LIN {X 0,Y 253.185,Z 308.196,A -85,B 0,C 180,E1 -19429.256,E2 -19429.256} C_VEL
LIN {X 0,Y 250.888,Z 304.72,A -85,B 0,C 180,E1 -19430.326,E2 -19430.326} C_VEL
LIN {X 0,Y 250.004,Z 303.462,A -85,B 0,C 180,E1 -19430.751,E2 -19430.751} C_VEL
LIN {X 0,Y 247.713,Z 300.458,A -85,B 0,C 180,E1 -19431.846,E2 -19431.846} C_VEL
LIN {X 0,Y 246.985,Z 298.947,A -85,B 0,C 180,E1 -19432.234,E2 -19432.234} C_VEL
LIN {X 0,Y 244.491,Z 296.754,A -85,B 0,C 180,E1 -19433.399,E2 -19433.399} C_VEL
LIN {X 0,Y 243.101,Z 294.193,A -85,B 0,C 180,E1 -19434.194,E2 -19434.194} C_VEL
LIN {X 0,Y 242.944,Z 293.571,A -85,B 0,C 180,E1 -19434.399,E2 -19434.399} C_VEL
LIN {X 0,Y 243.113,Z 292.905,A -85,B 0,C 180,E1 -19438.345,E2 -19438.345} C_VEL
LIN {X 0,Y 243.203,Z 292.718,A -85,B 0,C 180,E1 -19440.002,E2 -19440.002} C_VEL
LIN {X 0,Y 242.902,Z 292.579,A -85,B 0,C 180,E1 -19443.319,E2 -19443.319} C_VEL
LIN {X 0,Y 242.885,Z 292.698,A -85,B 0,C 180,E1 -19448.32,E2 -19448.32} C_VEL
LIN {X 0,Y 242.8,Z 293.112,A -85,B 0,C 180,E1 -19451.692,E2 -19451.692} C_VEL
LIN {X 0,Y 242.869,Z 293.758,A -85,B 0,C 180,E1 -19455.098,E2 -19455.098} C_VEL
LIN {X 0,Y 242.939,Z 294.698,A -85,B 0,C 180,E1 -19458.557,E2 -19458.557} C_VEL
LIN {X 0,Y 243.14,Z 296.031,A -85,B 0,C 180,E1 -19462.34,E2 -19462.34} C_VEL
LIN {X 0,Y 243.449,Z 297.883,A -85,B 0,C 180,E1 -19466.505,E2 -19466.505} C_VEL
LIN {X 0,Y 243.751,Z 299.841,A -85,B 0,C 180,E1 -19470.122,E2 -19470.122} C_VEL
LIN {X 0,Y 244.055,Z 301.816,A -85,B 0,C 180,E1 -19473.27,E2 -19473.27} C_VEL
LIN {X 0,Y 243.519,Z 302.82,A -85,B 0,C 180,E1 -19474.187,E2 -19474.187} C_VEL
LIN {X 0,Y 241.244,Z 305.585,A -85,B 0,C 180,E1 -19475.584,E2 -19475.584} C_VEL
LIN {X 0,Y 239.817,Z 308.232,A -85,B 0,C 180,E1 -19476.663,E2 -19476.663} C_VEL
LIN {X 0,Y 239.881,Z 310.193,A -85,B 0,C 180,E1 -19477.486,E2 -19477.486} C_VEL
LIN {X 0,Y 240.255,Z 310.779,A -85,B 0,C 180,E1 -19477.754,E2 -19477.754} C_VEL
LIN {X 0,Y 241.849,Z 312.454,A -85,B 0,C 180,E1 -19478.568,E2 -19478.568} C_VEL
LIN {X 0,Y 243.742,Z 316.37,A -85,B 0,C 180,E1 -19479.64,E2 -19479.64} C_VEL
LIN {X 0,Y 245.733,Z 319.174,A -85,B 0,C 180,E1 -19480.66,E2 -19480.66} C_VEL
LIN {X 0,Y 247.963,Z 323.482,A -85,B 0,C 180,E1 -19481.833,E2 -19481.833} C_VEL
LIN {X 0,Y 249.149,Z 325.386,A -85,B 0,C 180,E1 -19482.405,E2 -19482.405} C_VEL
LIN {X 0,Y 251.625,Z 330.796,A -85,B 0,C 180,E1 -19483.741,E2 -19483.741} C_VEL
LIN {X 0,Y 253.857,Z 336.868,A -85,B 0,C 180,E1 -19485.042,E2 -19485.042} C_VEL
LIN {X 0,Y 256.669,Z 347.947,A -85,B 0,C 180,E1 -19487.095,E2 -19487.095} C_VEL
LIN {X 0,Y 258.818,Z 360.728,A -85,B 0,C 180,E1 -19489.332,E2 -19489.332} C_VEL
LIN {X 0,Y 259.644,Z 370.662,A -85,B 0,C 180,E1 -19491.018,E2 -19491.018} C_VEL
LIN {X 0,Y 259.672,Z 381.634,A -85,B 0,C 180,E1 -19492.891,E2 -19492.891} C_VEL
LIN {X 0,Y 258.885,Z 392.631,A -85,B 0,C 180,E1 -19494.838,E2 -19494.838} C_VEL
LIN {X 0,Y 254.509,Z 405.491,A -85,B 0,C 180,E1 -19496.951,E2 -19496.951} C_VEL
LIN {X 0,Y 250.343,Z 416.596,A -85,B 0,C 180,E1 -19499.182,E2 -19499.182} C_VEL
LIN {X 0,Y 246.132,Z 427.508,A -85,B 0,C 180,E1 -19501.893,E2 -19501.893} C_VEL
LIN {X 0,Y 242.659,Z 436.647,A -85,B 0,C 180,E1 -19504.712,E2 -19504.712} C_VEL
LIN {X 0,Y 239.529,Z 444.307,A -85,B 0,C 180,E1 -19507.579,E2 -19507.579} C_VEL
LIN {X 0,Y 236.803,Z 451.549,A -85,B 0,C 180,E1 -19510.947,E2 -19510.947} C_VEL
LIN {X 0,Y 234.837,Z 457.354,A -85,B 0,C 180,E1 -19514.376,E2 -19514.376} C_VEL
LIN {X 0,Y 233.597,Z 461.841,A -85,B 0,C 180,E1 -19517.844,E2 -19517.844} C_VEL
LIN {X 0,Y 233.019,Z 465.103,A -85,B 0,C 180,E1 -19521.328,E2 -19521.328} C_VEL
LIN {X 0,Y 232.953,Z 467.185,A -85,B 0,C 180,E1 -19524.808,E2 -19524.808} C_VEL
LIN {X 0,Y 232.961,Z 468.034,A -85,B 0,C 180,E1 -19528.272,E2 -19528.272} C_VEL
LIN {X 0,Y 232.997,Z 468.019,A -85,B 0,C 180,E1 -19530.001,E2 -19530.001} C_VEL
LIN {X 0,Y 232.972,Z 467.09,A -85,B 0,C 180,E1 -19533.46,E2 -19533.46} C_VEL
LIN {X 0,Y 233.034,Z 465.926,A -85,B 0,C 180,E1 -19535.582,E2 -19535.582} C_VEL
LIN {X 0,Y 233.072,Z 463.412,A -85,B 0,C 180,E1 -19538.673,E2 -19538.673} C_VEL
LIN {X 0,Y 233.62,Z 459.368,A -85,B 0,C 180,E1 -19542.158,E2 -19542.158} C_VEL
LIN {X 0,Y 234.812,Z 453.934,A -85,B 0,C 180,E1 -19545.628,E2 -19545.628} C_VEL
LIN {X 0,Y 236.689,Z 446.986,A -85,B 0,C 180,E1 -19549.065,E2 -19549.065} C_VEL
LIN {X 0,Y 238.891,Z 439.482,A -85,B 0,C 180,E1 -19552.031,E2 -19552.031} C_VEL
LIN {X 0,Y 241.773,Z 430.492,A -85,B 0,C 180,E1 -19554.93,E2 -19554.93} C_VEL
LIN {X 0,Y 244.548,Z 421.312,A -85,B 0,C 180,E1 -19557.377,E2 -19557.377} C_VEL
LIN {X 0,Y 247.908,Z 410.531,A -85,B 0,C 180,E1 -19559.744,E2 -19559.744} C_VEL
LIN {X 0,Y 251.243,Z 398.782,A -85,B 0,C 180,E1 -19561.871,E2 -19561.871} C_VEL
LIN {X 0,Y 253.709,Z 390.137,A -85,B 0,C 180,E1 -19563.169,E2 -19563.169} C_VEL
LIN {X 0,Y 253.899,Z 385.833,A -85,B 0,C 180,E1 -19563.857,E2 -19563.857} C_VEL
LIN {X 0,Y 253.203,Z 373.399,A -85,B 0,C 180,E1 -19565.801,E2 -19565.801} C_VEL
LIN {X 0,Y 251.448,Z 358.938,A -85,B 0,C 180,E1 -19567.852,E2 -19567.852} C_VEL
LIN {X 0,Y 249.014,Z 346.189,A -85,B 0,C 180,E1 -19569.525,E2 -19569.525} C_VEL
LIN {X 0,Y 245.629,Z 332.569,A -85,B 0,C 180,E1 -19571.179,E2 -19571.179} C_VEL
LIN {X 0,Y 241.385,Z 319.106,A -85,B 0,C 180,E1 -19572.752,E2 -19572.752} C_VEL
LIN {X 0,Y 239.34,Z 314.218,A -85,B 0,C 180,E1 -19573.368,E2 -19573.368} C_VEL
LIN {X 0,Y 238.309,Z 310.845,A -85,B 0,C 180,E1 -19573.734,E2 -19573.734} C_VEL
LIN {X 0,Y 237.815,Z 307.272,A -85,B 0,C 180,E1 -19577.178,E2 -19577.178} C_VEL
LIN {X 0,Y 236.974,Z 303.106,A -85,B 0,C 180,E1 -19581.477,E2 -19581.477} C_VEL
LIN {X 0,Y 236.258,Z 298.657,A -85,B 0,C 180,E1 -19586.402,E2 -19586.402} C_VEL
LIN {X 0,Y 235.576,Z 294.467,A -85,B 0,C 180,E1 -19591.487,E2 -19591.487} C_VEL
LIN {X 0,Y 235.184,Z 291.61,A -85,B 0,C 180,E1 -19595.267,E2 -19595.267} C_VEL
LIN {X 0,Y 234.976,Z 290.842,A -85,B 0,C 180,E1 -19596.651,E2 -19596.651} C_VEL
LIN {X 0,Y 235.016,Z 290.835,A -85,B 0,C 180,E1 -19600.793,E2 -19600.793} C_VEL
LIN {X 0,Y 235.121,Z 290.825,A -85,B 0,C 180,E1 -19604.392,E2 -19604.392} C_VEL
LIN {X 0,Y 235.221,Z 290.812,A -85,B 0,C 180,E1 -19609.671,E2 -19609.671} C_VEL
LIN {X 0,Y 235.365,Z 290.793,A -85,B 0,C 180,E1 -19613.138,E2 -19613.138} C_VEL
LIN {X 0,Y 235.6,Z 290.764,A -85,B 0,C 180,E1 -19618.289,E2 -19618.289} C_VEL
LIN {X 0,Y 235.6,Z 290.761,A -85,B 0,C 180,E1 -19621.708,E2 -19621.708} C_VEL
LIN {X 0,Y 235.41,Z 290.784,A -85,B 0,C 180,E1 -19626.857,E2 -19626.857} C_VEL
LIN {X 0,Y 235.257,Z 290.798,A -85,B 0,C 180,E1 -19630.324,E2 -19630.324} C_VEL
LIN {X 0,Y 235.116,Z 290.82,A -85,B 0,C 180,E1 -19635.604,E2 -19635.604} C_VEL
LIN {X 0,Y 235.011,Z 290.825,A -85,B 0,C 180,E1 -19639.203,E2 -19639.203} C_VEL
LIN {X 0,Y 234.962,Z 290.84,A -85,B 0,C 180,E1 -19642.88,E2 -19642.88} C_VEL
LIN {X 0,Y 234.968,Z 290.832,A -85,B 0,C 180,E1 -19646.655,E2 -19646.655} C_VEL
LIN {X 0,Y 234.922,Z 290.845,A -85,B 0,C 180,E1 -19650.566,E2 -19650.566} C_VEL
LIN {X 0,Y 234.959,Z 290.832,A -85,B 0,C 180,E1 -19654.63,E2 -19654.63} C_VEL
LIN {X 0,Y 234.94,Z 290.843,A -85,B 0,C 180,E1 -19658.942,E2 -19658.942} C_VEL
LIN {X 0,Y 234.901,Z 290.836,A -85,B 0,C 180,E1 -19663.48,E2 -19663.48} C_VEL
LIN {X 0,Y 234.962,Z 290.841,A -85,B 0,C 180,E1 -19666.53,E2 -19666.53} C_VEL
LIN {X 0,Y 234.951,Z 290.84,A -85,B 0,C 180,E1 -19671.084,E2 -19671.084} C_VEL
LIN {X 0,Y 234.955,Z 290.834,A -85,B 0,C 180,E1 -19675.365,E2 -19675.365} C_VEL
LIN {X 0,Y 234.964,Z 290.836,A -85,B 0,C 180,E1 -19680.155,E2 -19680.155} C_VEL
LIN {X 0,Y 234.988,Z 290.838,A -85,B 0,C 180,E1 -19683.791,E2 -19683.791} C_VEL
LIN {X 0,Y 235.004,Z 290.833,A -85,B 0,C 180,E1 -19688.968,E2 -19688.968} C_VEL
LIN {X 0,Y 235.089,Z 290.822,A -85,B 0,C 180,E1 -19693.058,E2 -19693.058} C_VEL
LIN {X 0,Y 235.139,Z 290.818,A -85,B 0,C 180,E1 -19697.922,E2 -19697.922} C_VEL
LIN {X 0,Y 235.194,Z 290.863,A -85,B 0,C 180,E1 -19699.252,E2 -19699.252} C_VEL
LIN {X 0,Y 236.19,Z 293.619,A -85,B 0,C 180,E1 -19699.592,E2 -19699.592} C_VEL
LIN {X 0,Y 237.987,Z 295.971,A -85,B 0,C 180,E1 -19700.061,E2 -19700.061} C_VEL
LIN {X 0,Y 243.806,Z 306.338,A -85,B 0,C 180,E1 -19701.824,E2 -19701.824} C_VEL
LIN {X 0,Y 250.316,Z 320.248,A -85,B 0,C 180,E1 -19704.118,E2 -19704.118} C_VEL
LIN {X 0,Y 253.968,Z 333.092,A -85,B 0,C 180,E1 -19706.058,E2 -19706.058} C_VEL
LIN {X 0,Y 256.518,Z 342.604,A -85,B 0,C 180,E1 -19707.638,E2 -19707.638} C_VEL
LIN {X 0,Y 257.848,Z 349.694,A -85,B 0,C 180,E1 -19708.828,E2 -19708.828} C_VEL
LIN {X 0,Y 254.793,Z 363.082,A -85,B 0,C 180,E1 -19710.592,E2 -19710.592} C_VEL
LIN {X 0,Y 251.546,Z 375.487,A -85,B 0,C 180,E1 -19712.6,E2 -19712.6} C_VEL
LIN {X 0,Y 248.374,Z 386.892,A -85,B 0,C 180,E1 -19714.868,E2 -19714.868} C_VEL
LIN {X 0,Y 245.142,Z 397.448,A -85,B 0,C 180,E1 -19717.411,E2 -19717.411} C_VEL
LIN {X 0,Y 242.266,Z 406.393,A -85,B 0,C 180,E1 -19720.023,E2 -19720.023} C_VEL
LIN {X 0,Y 239.466,Z 415.098,A -85,B 0,C 180,E1 -19723.146,E2 -19723.146} C_VEL
LIN {X 0,Y 237.263,Z 422.246,A -85,B 0,C 180,E1 -19726.343,E2 -19726.343} C_VEL
LIN {X 0,Y 235.72,Z 427.315,A -85,B 0,C 180,E1 -19729.144,E2 -19729.144} C_VEL
LIN {X 0,Y 234.633,Z 431.161,A -85,B 0,C 180,E1 -19731.797,E2 -19731.797} C_VEL
LIN {X 0,Y 233.572,Z 435.229,A -85,B 0,C 180,E1 -19735.494,E2 -19735.494} C_VEL
LIN {X 0,Y 232.973,Z 437.791,A -85,B 0,C 180,E1 -19738.98,E2 -19738.98} C_VEL
LIN {X 0,Y 232.765,Z 439.248,A -85,B 0,C 180,E1 -19742.919,E2 -19742.919} C_VEL
LIN {X 0,Y 232.885,Z 439.402,A -85,B 0,C 180,E1 -19745.436,E2 -19745.436} C_VEL
LIN {X 0,Y 233.412,Z 438.539,A -85,B 0,C 180,E1 -19749.219,E2 -19749.219} C_VEL
LIN {X 0,Y 233.949,Z 437.448,A -85,B 0,C 180,E1 -19751.366,E2 -19751.366} C_VEL
LIN {X 0,Y 234.921,Z 435.417,A -85,B 0,C 180,E1 -19754.114,E2 -19754.114} C_VEL
LIN {X 0,Y 236.788,Z 431.27,A -85,B 0,C 180,E1 -19757.901,E2 -19757.901} C_VEL
LIN {X 0,Y 238.907,Z 426.574,A -85,B 0,C 180,E1 -19761.041,E2 -19761.041} C_VEL
LIN {X 0,Y 241.891,Z 419.933,A -85,B 0,C 180,E1 -19764.476,E2 -19764.476} C_VEL
LIN {X 0,Y 245.485,Z 411.83,A -85,B 0,C 180,E1 -19767.733,E2 -19767.733} C_VEL
LIN {X 0,Y 248.949,Z 403.623,A -85,B 0,C 180,E1 -19770.373,E2 -19770.373} C_VEL
LIN {X 0,Y 252.728,Z 394.225,A -85,B 0,C 180,E1 -19772.855,E2 -19772.855} C_VEL
LIN {X 0,Y 256.721,Z 383.792,A -85,B 0,C 180,E1 -19775.106,E2 -19775.106} C_VEL
LIN {X 0,Y 260.797,Z 371.812,A -85,B 0,C 180,E1 -19777.231,E2 -19777.231} C_VEL
LIN {X 0,Y 264.722,Z 358.953,A -85,B 0,C 180,E1 -19779.064,E2 -19779.064} C_VEL
LIN {X 0,Y 265.019,Z 357.032,A -85,B 0,C 180,E1 -19779.365,E2 -19779.365} C_VEL
LIN {X 0,Y 263.431,Z 347.65,A -85,B 0,C 180,E1 -19781.33,E2 -19781.33} C_VEL
LIN {X 0,Y 260.707,Z 337.459,A -85,B 0,C 180,E1 -19783.559,E2 -19783.559} C_VEL
LIN {X 0,Y 257.233,Z 328.172,A -85,B 0,C 180,E1 -19785.767,E2 -19785.767} C_VEL
LIN {X 0,Y 253.496,Z 320.497,A -85,B 0,C 180,E1 -19787.823,E2 -19787.823} C_VEL
LIN {X 0,Y 249.727,Z 313.921,A -85,B 0,C 180,E1 -19789.799,E2 -19789.799} C_VEL
LIN {X 0,Y 247.455,Z 310.146,A -85,B 0,C 180,E1 -19791.026,E2 -19791.026} C_VEL
LIN {X 0,Y 244.652,Z 306.273,A -85,B 0,C 180,E1 -19792.471,E2 -19792.471} C_VEL
LIN {X 0,Y 243.776,Z 304.918,A -85,B 0,C 180,E1 -19792.964,E2 -19792.964} C_VEL
LIN {X 0,Y 241.494,Z 302.282,A -85,B 0,C 180,E1 -19794.208,E2 -19794.208} C_VEL
LIN {X 0,Y 240.221,Z 300.054,A -85,B 0,C 180,E1 -19794.967,E2 -19794.967} C_VEL
LIN {X 0,Y 237.566,Z 297.828,A -85,B 0,C 180,E1 -19796.451,E2 -19796.451} C_VEL
LIN {X 0,Y 236.246,Z 295.17,A -85,B 0,C 180,E1 -19797.391,E2 -19797.391} C_VEL
LIN {X 0,Y 236.11,Z 294.602,A -85,B 0,C 180,E1 -19797.55,E2 -19797.55} C_VEL
LIN {X 0,Y 236.297,Z 294.313,A -85,B 0,C 180,E1 -19800.002,E2 -19800.002} C_VEL
LIN {X 0,Y 235.978,Z 294.218,A -85,B 0,C 180,E1 -19803.417,E2 -19803.417} C_VEL
LIN {X 0,Y 235.991,Z 294.39,A -85,B 0,C 180,E1 -19808.565,E2 -19808.565} C_VEL
LIN {X 0,Y 235.907,Z 294.845,A -85,B 0,C 180,E1 -19812.039,E2 -19812.039} C_VEL
LIN {X 0,Y 235.977,Z 295.543,A -85,B 0,C 180,E1 -19815.55,E2 -19815.55} C_VEL
LIN {X 0,Y 236.04,Z 296.55,A -85,B 0,C 180,E1 -19819.12,E2 -19819.12} C_VEL
LIN {X 0,Y 236.262,Z 297.852,A -85,B 0,C 180,E1 -19822.762,E2 -19822.762} C_VEL
LIN {X 0,Y 236.586,Z 299.74,A -85,B 0,C 180,E1 -19826.982,E2 -19826.982} C_VEL
LIN {X 0,Y 236.851,Z 301.727,A -85,B 0,C 180,E1 -19830.629,E2 -19830.629} C_VEL
LIN {X 0,Y 237.356,Z 304.683,A -85,B 0,C 180,E1 -19835.268,E2 -19835.268} C_VEL
LIN {X 0,Y 237.427,Z 305.216,A -85,B 0,C 180,E1 -19835.974,E2 -19835.974} C_VEL
LIN {X 0,Y 238.662,Z 308.471,A -85,B 0,C 180,E1 -19836.828,E2 -19836.828} C_VEL
LIN {X 0,Y 240.255,Z 310.779,A -85,B 0,C 180,E1 -19837.754,E2 -19837.754} C_VEL
LIN {X 0,Y 241.412,Z 313.155,A -85,B 0,C 180,E1 -19838.442,E2 -19838.442} C_VEL
LIN {X 0,Y 242.047,Z 316.408,A -85,B 0,C 180,E1 -19838.976,E2 -19838.976} C_VEL
LIN {X 0,Y 242.792,Z 324.718,A -85,B 0,C 180,E1 -19840.101,E2 -19840.101} C_VEL
LIN {X 0,Y 243.621,Z 327.601,A -85,B 0,C 180,E1 -19840.744,E2 -19840.744} C_VEL
LIN {X 0,Y 245.539,Z 331.037,A -85,B 0,C 180,E1 -19841.802,E2 -19841.802} C_VEL
LIN {X 0,Y 247.719,Z 336.19,A -85,B 0,C 180,E1 -19843.129,E2 -19843.129} C_VEL
LIN {X 0,Y 249.241,Z 340.665,A -85,B 0,C 180,E1 -19844.139,E2 -19844.139} C_VEL
LIN {X 0,Y 251.691,Z 351.39,A -85,B 0,C 180,E1 -19846.263,E2 -19846.263} C_VEL
LIN {X 0,Y 253.409,Z 363.466,A -85,B 0,C 180,E1 -19848.489,E2 -19848.489} C_VEL
LIN {X 0,Y 253.991,Z 373.209,A -85,B 0,C 180,E1 -19850.245,E2 -19850.245} C_VEL
LIN {X 0,Y 253.768,Z 384.036,A -85,B 0,C 180,E1 -19852.196,E2 -19852.196} C_VEL
LIN {X 0,Y 252.88,Z 393.443,A -85,B 0,C 180,E1 -19853.949,E2 -19853.949} C_VEL
LIN {X 0,Y 250.951,Z 399.558,A -85,B 0,C 180,E1 -19854.964,E2 -19854.964} C_VEL
LIN {X 0,Y 246.385,Z 411.496,A -85,B 0,C 180,E1 -19857.184,E2 -19857.184} C_VEL
LIN {X 0,Y 242.295,Z 421.625,A -85,B 0,C 180,E1 -19859.497,E2 -19859.497} C_VEL
LIN {X 0,Y 238.221,Z 431.45,A -85,B 0,C 180,E1 -19862.261,E2 -19862.261} C_VEL
LIN {X 0,Y 234.777,Z 439.999,A -85,B 0,C 180,E1 -19865.224,E2 -19865.224} C_VEL
LIN {X 0,Y 232.122,Z 446.12,A -85,B 0,C 180,E1 -19867.763,E2 -19867.763} C_VEL
LIN {X 0,Y 229.422,Z 452.928,A -85,B 0,C 180,E1 -19871.239,E2 -19871.239} C_VEL
LIN {X 0,Y 227.53,Z 458.343,A -85,B 0,C 180,E1 -19874.78,E2 -19874.78} C_VEL
LIN {X 0,Y 226.591,Z 461.52,A -85,B 0,C 180,E1 -19877.462,E2 -19877.462} C_VEL
LIN {X 0,Y 225.952,Z 464.735,A -85,B 0,C 180,E1 -19881.054,E2 -19881.054} C_VEL
LIN {X 0,Y 225.886,Z 466.782,A -85,B 0,C 180,E1 -19884.646,E2 -19884.646} C_VEL
LIN {X 0,Y 225.892,Z 467.604,A -85,B 0,C 180,E1 -19888.218,E2 -19888.218} C_VEL
LIN {X 0,Y 225.925,Z 467.565,A -85,B 0,C 180,E1 -19890.001,E2 -19890.001} C_VEL
LIN {X 0,Y 225.891,Z 466.591,A -85,B 0,C 180,E1 -19893.569,E2 -19893.569} C_VEL
LIN {X 0,Y 225.955,Z 465.543,A -85,B 0,C 180,E1 -19895.536,E2 -19895.536} C_VEL
LIN {X 0,Y 225.999,Z 462.839,A -85,B 0,C 180,E1 -19898.946,E2 -19898.946} C_VEL
LIN {X 0,Y 226.618,Z 458.742,A -85,B 0,C 180,E1 -19902.539,E2 -19902.539} C_VEL
LIN {X 0,Y 227.907,Z 453.259,A -85,B 0,C 180,E1 -19906.114,E2 -19906.114} C_VEL
LIN {X 0,Y 229.903,Z 446.243,A -85,B 0,C 180,E1 -19909.651,E2 -19909.651} C_VEL
LIN {X 0,Y 232.252,Z 438.698,A -85,B 0,C 180,E1 -19912.696,E2 -19912.696} C_VEL
LIN {X 0,Y 235.271,Z 429.633,A -85,B 0,C 180,E1 -19915.668,E2 -19915.668} C_VEL
LIN {X 0,Y 238.179,Z 420.367,A -85,B 0,C 180,E1 -19918.173,E2 -19918.173} C_VEL
LIN {X 0,Y 241.695,Z 409.488,A -85,B 0,C 180,E1 -19920.589,E2 -19920.589} C_VEL
LIN {X 0,Y 245.153,Z 397.616,A -85,B 0,C 180,E1 -19922.76,E2 -19922.76} C_VEL
LIN {X 0,Y 247.384,Z 389.587,A -85,B 0,C 180,E1 -19923.997,E2 -19923.997} C_VEL
LIN {X 0,Y 247.01,Z 378.181,A -85,B 0,C 180,E1 -19925.907,E2 -19925.907} C_VEL
LIN {X 0,Y 245.862,Z 365.767,A -85,B 0,C 180,E1 -19927.82,E2 -19927.82} C_VEL
LIN {X 0,Y 243.985,Z 353.362,A -85,B 0,C 180,E1 -19929.569,E2 -19929.569} C_VEL
LIN {X 0,Y 240.901,Z 339.012,A -85,B 0,C 180,E1 -19931.46,E2 -19931.46} C_VEL
LIN {X 0,Y 236.907,Z 325.205,A -85,B 0,C 180,E1 -19933.207,E2 -19933.207} C_VEL
LIN {X 0,Y 234.045,Z 317.638,A -85,B 0,C 180,E1 -19934.181,E2 -19934.181} C_VEL
LIN {X 0,Y 232.658,Z 314.388,A -85,B 0,C 180,E1 -19934.615,E2 -19934.615} C_VEL
LIN {X 0,Y 231.327,Z 311.19,A -85,B 0,C 180,E1 -19935.032,E2 -19935.032} C_VEL
LIN {X 0,Y 231.187,Z 310.338,A -85,B 0,C 180,E1 -19935.14,E2 -19935.14} C_VEL
LIN {X 0,Y 230.316,Z 305.901,A -85,B 0,C 180,E1 -19939.719,E2 -19939.719} C_VEL
LIN {X 0,Y 229.496,Z 301.644,A -85,B 0,C 180,E1 -19944.418,E2 -19944.418} C_VEL
LIN {X 0,Y 228.95,Z 298.172,A -85,B 0,C 180,E1 -19948.542,E2 -19948.542} C_VEL
LIN {X 0,Y 228.429,Z 294.593,A -85,B 0,C 180,E1 -19953.157,E2 -19953.157} C_VEL
LIN {X 0,Y 227.951,Z 291.717,A -85,B 0,C 180,E1 -19957.494,E2 -19957.494} C_VEL
LIN {X 0,Y 228.042,Z 291.707,A -85,B 0,C 180,E1 -19962.824,E2 -19962.824} C_VEL
LIN {X 0,Y 228.079,Z 291.702,A -85,B 0,C 180,E1 -19967.542,E2 -19967.542} C_VEL
LIN {X 0,Y 228.265,Z 291.679,A -85,B 0,C 180,E1 -19971.143,E2 -19971.143} C_VEL
LIN {X 0,Y 228.317,Z 291.672,A -85,B 0,C 180,E1 -19972.926,E2 -19972.926} C_VEL
LIN {X 0,Y 228.558,Z 291.641,A -85,B 0,C 180,E1 -19978.236,E2 -19978.236} C_VEL
LIN {X 0,Y 228.559,Z 291.638,A -85,B 0,C 180,E1 -19981.76,E2 -19981.76} C_VEL
LIN {X 0,Y 228.362,Z 291.662,A -85,B 0,C 180,E1 -19987.069,E2 -19987.069} C_VEL
LIN {X 0,Y 228.171,Z 291.678,A -85,B 0,C 180,E1 -19990.648,E2 -19990.648} C_VEL
LIN {X 0,Y 228.068,Z 291.694,A -85,B 0,C 180,E1 -19994.27,E2 -19994.27} C_VEL
LIN {X 0,Y 228.006,Z 291.703,A -85,B 0,C 180,E1 -19997.951,E2 -19997.951} C_VEL
LIN {X 0,Y 227.932,Z 291.712,A -85,B 0,C 180,E1 -20002.327,E2 -20002.327} C_VEL
LIN {X 0,Y 227.942,Z 291.707,A -85,B 0,C 180,E1 -20006.6,E2 -20006.6} C_VEL
LIN {X 0,Y 227.897,Z 291.717,A -85,B 0,C 180,E1 -20010.289,E2 -20010.289} C_VEL
LIN {X 0,Y 227.889,Z 291.719,A -85,B 0,C 180,E1 -20013.716,E2 -20013.716} C_VEL
LIN {X 0,Y 227.868,Z 291.723,A -85,B 0,C 180,E1 -20018.083,E2 -20018.083} C_VEL
LIN {X 0,Y 227.835,Z 291.714,A -85,B 0,C 180,E1 -20022.733,E2 -20022.733} C_VEL
LIN {X 0,Y 227.906,Z 291.721,A -85,B 0,C 180,E1 -20027.278,E2 -20027.278} C_VEL
LIN {X 0,Y 227.867,Z 291.727,A -85,B 0,C 180,E1 -20031.912,E2 -20031.912} C_VEL
LIN {X 0,Y 227.885,Z 291.722,A -85,B 0,C 180,E1 -20036.371,E2 -20036.371} C_VEL
LIN {X 0,Y 227.914,Z 291.714,A -85,B 0,C 180,E1 -20040.436,E2 -20040.436} C_VEL
LIN {X 0,Y 227.922,Z 291.715,A -85,B 0,C 180,E1 -20044.424,E2 -20044.424} C_VEL
LIN {X 0,Y 227.955,Z 291.713,A -85,B 0,C 180,E1 -20048.285,E2 -20048.285} C_VEL
LIN {X 0,Y 228.027,Z 291.7,A -85,B 0,C 180,E1 -20052.824,E2 -20052.824} C_VEL
LIN {X 0,Y 228.104,Z 291.695,A -85,B 0,C 180,E1 -20057.826,E2 -20057.826} C_VEL
LIN {X 0,Y 229.182,Z 294.671,A -85,B 0,C 180,E1 -20058.236,E2 -20058.236} C_VEL
LIN {X 0,Y 230.91,Z 296.956,A -85,B 0,C 180,E1 -20058.716,E2 -20058.716} C_VEL
LIN {X 0,Y 232.983,Z 300.19,A -85,B 0,C 180,E1 -20059.35,E2 -20059.35} C_VEL
LIN {X 0,Y 238.48,Z 310.065,A -85,B 0,C 180,E1 -20061.144,E2 -20061.144} C_VEL
LIN {X 0,Y 244.812,Z 324.149,A -85,B 0,C 180,E1 -20063.588,E2 -20063.588} C_VEL
LIN {X 0,Y 248.362,Z 337.496,A -85,B 0,C 180,E1 -20065.739,E2 -20065.739} C_VEL
LIN {X 0,Y 250.92,Z 347.895,A -85,B 0,C 180,E1 -20067.563,E2 -20067.563} C_VEL
LIN {X 0,Y 251.488,Z 351.022,A -85,B 0,C 180,E1 -20068.121,E2 -20068.121} C_VEL
LIN {X 0,Y 248.25,Z 364.738,A -85,B 0,C 180,E1 -20069.999,E2 -20069.999} C_VEL
LIN {X 0,Y 244.966,Z 376.908,A -85,B 0,C 180,E1 -20072.054,E2 -20072.054} C_VEL
LIN {X 0,Y 241.96,Z 387.219,A -85,B 0,C 180,E1 -20074.163,E2 -20074.163} C_VEL
LIN {X 0,Y 238.598,Z 397.796,A -85,B 0,C 180,E1 -20076.765,E2 -20076.765} C_VEL
LIN {X 0,Y 235.302,Z 407.631,A -85,B 0,C 180,E1 -20079.736,E2 -20079.736} C_VEL
LIN {X 0,Y 232.334,Z 416.483,A -85,B 0,C 180,E1 -20083.069,E2 -20083.069} C_VEL
LIN {X 0,Y 230.377,Z 422.64,A -85,B 0,C 180,E1 -20085.934,E2 -20085.934} C_VEL
LIN {X 0,Y 228.767,Z 427.72,A -85,B 0,C 180,E1 -20088.822,E2 -20088.822} C_VEL
LIN {X 0,Y 227.444,Z 432.17,A -85,B 0,C 180,E1 -20092.035,E2 -20092.035} C_VEL
LIN {X 0,Y 226.402,Z 436.039,A -85,B 0,C 180,E1 -20095.819,E2 -20095.819} C_VEL
LIN {X 0,Y 225.772,Z 438.668,A -85,B 0,C 180,E1 -20099.87,E2 -20099.87} C_VEL
LIN {X 0,Y 225.697,Z 439.661,A -85,B 0,C 180,E1 -20102.785,E2 -20102.785} C_VEL
LIN {X 0,Y 225.863,Z 439.831,A -85,B 0,C 180,E1 -20106.241,E2 -20106.241} C_VEL
LIN {X 0,Y 226.3,Z 439.182,A -85,B 0,C 180,E1 -20109.072,E2 -20109.072} C_VEL
LIN {X 0,Y 227.342,Z 437.219,A -85,B 0,C 180,E1 -20112.85,E2 -20112.85} C_VEL
LIN {X 0,Y 228.748,Z 434.341,A -85,B 0,C 180,E1 -20116.219,E2 -20116.219} C_VEL
LIN {X 0,Y 230.774,Z 430.263,A -85,B 0,C 180,E1 -20119.581,E2 -20119.581} C_VEL
LIN {X 0,Y 233.31,Z 424.892,A -85,B 0,C 180,E1 -20122.957,E2 -20122.957} C_VEL
LIN {X 0,Y 236.581,Z 418.054,A -85,B 0,C 180,E1 -20126.28,E2 -20126.28} C_VEL
LIN {X 0,Y 240.483,Z 409.509,A -85,B 0,C 180,E1 -20129.553,E2 -20129.553} C_VEL
LIN {X 0,Y 244.313,Z 400.922,A -85,B 0,C 180,E1 -20132.185,E2 -20132.185} C_VEL
LIN {X 0,Y 248.612,Z 390.578,A -85,B 0,C 180,E1 -20134.767,E2 -20134.767} C_VEL
LIN {X 0,Y 253.087,Z 378.843,A -85,B 0,C 180,E1 -20137.124,E2 -20137.124} C_VEL
LIN {X 0,Y 257.059,Z 367.185,A -85,B 0,C 180,E1 -20139.031,E2 -20139.031} C_VEL
LIN {X 0,Y 259.151,Z 360.42,A -85,B 0,C 180,E1 -20139.98,E2 -20139.98} C_VEL
LIN {X 0,Y 259.066,Z 357.445,A -85,B 0,C 180,E1 -20140.592,E2 -20140.592} C_VEL
LIN {X 0,Y 257.319,Z 347.685,A -85,B 0,C 180,E1 -20142.769,E2 -20142.769} C_VEL
LIN {X 0,Y 254.435,Z 337.495,A -85,B 0,C 180,E1 -20145.214,E2 -20145.214} C_VEL
LIN {X 0,Y 251.007,Z 328.913,A -85,B 0,C 180,E1 -20147.486,E2 -20147.486} C_VEL
LIN {X 0,Y 246.298,Z 319.735,A -85,B 0,C 180,E1 -20150.296,E2 -20150.296} C_VEL
LIN {X 0,Y 244.08,Z 315.885,A -85,B 0,C 180,E1 -20151.618,E2 -20151.618} C_VEL
LIN {X 0,Y 241.448,Z 311.907,A -85,B 0,C 180,E1 -20153.158,E2 -20153.158} C_VEL
LIN {X 0,Y 238.316,Z 307.697,A -85,B 0,C 180,E1 -20155.038,E2 -20155.038} C_VEL
LIN {X 0,Y 237.457,Z 306.358,A -85,B 0,C 180,E1 -20155.602,E2 -20155.602} C_VEL
LIN {X 0,Y 234.961,Z 303.676,A -85,B 0,C 180,E1 -20157.216,E2 -20157.216} C_VEL
LIN {X 0,Y 233.696,Z 301.169,A -85,B 0,C 180,E1 -20158.171,E2 -20158.171} C_VEL
LIN {X 0,Y 231.222,Z 299.31,A -85,B 0,C 180,E1 -20159.894,E2 -20159.894} C_VEL
LIN {X 0,Y 229.62,Z 296.935,A -85,B 0,C 180,E1 -20161.262,E2 -20161.262} C_VEL
LIN {X 0,Y 229.27,Z 295.841,A -85,B 0,C 180,E1 -20161.649,E2 -20161.649} C_VEL
LIN {X 0,Y 229.036,Z 295.952,A -85,B 0,C 180,E1 -20167.052,E2 -20167.052} C_VEL
LIN {X 0,Y 229.025,Z 296.339,A -85,B 0,C 180,E1 -20170.903,E2 -20170.903} C_VEL
LIN {X 0,Y 229.093,Z 297.353,A -85,B 0,C 180,E1 -20176.029,E2 -20176.029} C_VEL
LIN {X 0,Y 229.168,Z 298.425,A -85,B 0,C 180,E1 -20179.717,E2 -20179.717} C_VEL
LIN {X 0,Y 229.391,Z 299.801,A -85,B 0,C 180,E1 -20183.473,E2 -20183.473} C_VEL
LIN {X 0,Y 229.696,Z 301.604,A -85,B 0,C 180,E1 -20187.466,E2 -20187.466} C_VEL
LIN {X 0,Y 230.026,Z 303.953,A -85,B 0,C 180,E1 -20191.679,E2 -20191.679} C_VEL
LIN {X 0,Y 231.239,Z 307.164,A -85,B 0,C 180,E1 -20192.779,E2 -20192.779} C_VEL
LIN {X 0,Y 234.077,Z 310.745,A -85,B 0,C 180,E1 -20194.784,E2 -20194.784} C_VEL
LIN {X 0,Y 234.895,Z 311.647,A -85,B 0,C 180,E1 -20195.299,E2 -20195.299} C_VEL
LIN {X 0,Y 236.555,Z 315.262,A -85,B 0,C 180,E1 -20196.457,E2 -20196.457} C_VEL
LIN {X 0,Y 238.992,Z 318.69,A -85,B 0,C 180,E1 -20197.947,E2 -20197.947} C_VEL
LIN {X 0,Y 241.058,Z 322.792,A -85,B 0,C 180,E1 -20199.221,E2 -20199.221} C_VEL
LIN {X 0,Y 242.493,Z 324.999,A -85,B 0,C 180,E1 -20200.021,E2 -20200.021} C_VEL
LIN {X 0,Y 243.621,Z 327.601,A -85,B 0,C 180,E1 -20200.744,E2 -20200.744} C_VEL
LIN {X 0,Y 245.074,Z 331.601,A -85,B 0,C 180,E1 -20201.705,E2 -20201.705} C_VEL
LIN {X 0,Y 245.807,Z 336.367,A -85,B 0,C 180,E1 -20202.521,E2 -20202.521} C_VEL
LIN {X 0,Y 246.13,Z 350.091,A -85,B 0,C 180,E1 -20204.518,E2 -20204.518} C_VEL
LIN {X 0,Y 246.451,Z 353.274,A -85,B 0,C 180,E1 -20205.097,E2 -20205.097} C_VEL
LIN {X 0,Y 247.967,Z 365.366,A -85,B 0,C 180,E1 -20207.47,E2 -20207.47} C_VEL
LIN {X 0,Y 248.373,Z 375.469,A -85,B 0,C 180,E1 -20209.399,E2 -20209.399} C_VEL
LIN {X 0,Y 247.914,Z 386.135,A -85,B 0,C 180,E1 -20211.417,E2 -20211.417} C_VEL
LIN {X 0,Y 246.747,Z 395.546,A -85,B 0,C 180,E1 -20213.265,E2 -20213.265} C_VEL
LIN {X 0,Y 242.759,Z 406.075,A -85,B 0,C 180,E1 -20215.128,E2 -20215.128} C_VEL
LIN {X 0,Y 238.253,Z 416.932,A -85,B 0,C 180,E1 -20217.431,E2 -20217.431} C_VEL
LIN {X 0,Y 233.618,Z 427.591,A -85,B 0,C 180,E1 -20220.241,E2 -20220.241} C_VEL
LIN {X 0,Y 229.748,Z 436.558,A -85,B 0,C 180,E1 -20223.181,E2 -20223.181} C_VEL
LIN {X 0,Y 226.326,Z 444.082,A -85,B 0,C 180,E1 -20226.193,E2 -20226.193} C_VEL
LIN {X 0,Y 223.275,Z 451.182,A -85,B 0,C 180,E1 -20229.744,E2 -20229.744} C_VEL
LIN {X 0,Y 221.051,Z 456.849,A -85,B 0,C 180,E1 -20233.374,E2 -20233.374} C_VEL
LIN {X 0,Y 219.598,Z 461.216,A -85,B 0,C 180,E1 -20237.056,E2 -20237.056} C_VEL
LIN {X 0,Y 218.903,Z 464.373,A -85,B 0,C 180,E1 -20240.764,E2 -20240.764} C_VEL
LIN {X 0,Y 218.787,Z 466.46,A -85,B 0,C 180,E1 -20244.759,E2 -20244.759} C_VEL
LIN {X 0,Y 218.823,Z 467.175,A -85,B 0,C 180,E1 -20248.161,E2 -20248.161} C_VEL
LIN {X 0,Y 218.855,Z 467.114,A -85,B 0,C 180,E1 -20250.001,E2 -20250.001} C_VEL
LIN {X 0,Y 218.813,Z 466.091,A -85,B 0,C 180,E1 -20253.684,E2 -20253.684} C_VEL
LIN {X 0,Y 218.891,Z 465.132,A -85,B 0,C 180,E1 -20255.529,E2 -20255.529} C_VEL
LIN {X 0,Y 218.946,Z 462.261,A -85,B 0,C 180,E1 -20259.237,E2 -20259.237} C_VEL
LIN {X 0,Y 219.624,Z 458.109,A -85,B 0,C 180,E1 -20262.945,E2 -20262.945} C_VEL
LIN {X 0,Y 221.016,Z 452.568,A -85,B 0,C 180,E1 -20266.631,E2 -20266.631} C_VEL
LIN {X 0,Y 223.14,Z 445.489,A -85,B 0,C 180,E1 -20270.272,E2 -20270.272} C_VEL
LIN {X 0,Y 225.649,Z 437.907,A -85,B 0,C 180,E1 -20273.399,E2 -20273.399} C_VEL
LIN {X 0,Y 228.788,Z 428.77,A -85,B 0,C 180,E1 -20276.451,E2 -20276.451} C_VEL
LIN {X 0,Y 231.848,Z 419.421,A -85,B 0,C 180,E1 -20279.014,E2 -20279.014} C_VEL
LIN {X 0,Y 235.542,Z 408.447,A -85,B 0,C 180,E1 -20281.478,E2 -20281.478} C_VEL
LIN {X 0,Y 238.782,Z 397.628,A -85,B 0,C 180,E1 -20283.496,E2 -20283.496} C_VEL
LIN {X 0,Y 240.661,Z 391.668,A -85,B 0,C 180,E1 -20284.435,E2 -20284.435} C_VEL
LIN {X 0,Y 240.728,Z 383.194,A -85,B 0,C 180,E1 -20285.933,E2 -20285.933} C_VEL
LIN {X 0,Y 239.827,Z 369.804,A -85,B 0,C 180,E1 -20288.128,E2 -20288.128} C_VEL
LIN {X 0,Y 238.312,Z 357.887,A -85,B 0,C 180,E1 -20289.934,E2 -20289.934} C_VEL
LIN {X 0,Y 235.314,Z 342.474,A -85,B 0,C 180,E1 -20292.113,E2 -20292.113} C_VEL
LIN {X 0,Y 231.574,Z 328.725,A -85,B 0,C 180,E1 -20293.958,E2 -20293.958} C_VEL
LIN {X 0,Y 228.007,Z 318.987,A -85,B 0,C 180,E1 -20295.298,E2 -20295.298} C_VEL
LIN {X 0,Y 225.81,Z 314.381,A -85,B 0,C 180,E1 -20296.001,E2 -20296.001} C_VEL
LIN {X 0,Y 224.252,Z 311.473,A -85,B 0,C 180,E1 -20296.487,E2 -20296.487} C_VEL
LIN {X 0,Y 223.869,Z 309.818,A -85,B 0,C 180,E1 -20296.704,E2 -20296.704} C_VEL
LIN {X 0,Y 223.033,Z 305.915,A -85,B 0,C 180,E1 -20300.932,E2 -20300.932} C_VEL
LIN {X 0,Y 222.397,Z 302.102,A -85,B 0,C 180,E1 -20305.33,E2 -20305.33} C_VEL
LIN {X 0,Y 221.85,Z 298.694,A -85,B 0,C 180,E1 -20309.543,E2 -20309.543} C_VEL
LIN {X 0,Y 221.408,Z 295.645,A -85,B 0,C 180,E1 -20313.614,E2 -20313.614} C_VEL
LIN {X 0,Y 220.94,Z 292.589,A -85,B 0,C 180,E1 -20318.296,E2 -20318.296} C_VEL
LIN {X 0,Y 221.023,Z 292.58,A -85,B 0,C 180,E1 -20323.369,E2 -20323.369} C_VEL
LIN {X 0,Y 221.088,Z 292.574,A -85,B 0,C 180,E1 -20329.003,E2 -20329.003} C_VEL
LIN {X 0,Y 221.253,Z 292.553,A -85,B 0,C 180,E1 -20332.699,E2 -20332.699} C_VEL
LIN {X 0,Y 221.516,Z 292.518,A -85,B 0,C 180,E1 -20338.18,E2 -20338.18} C_VEL
LIN {X 0,Y 221.517,Z 292.516,A -85,B 0,C 180,E1 -20341.816,E2 -20341.816} C_VEL
LIN {X 0,Y 221.315,Z 292.539,A -85,B 0,C 180,E1 -20347.296,E2 -20347.296} C_VEL
LIN {X 0,Y 221.115,Z 292.555,A -85,B 0,C 180,E1 -20350.992,E2 -20350.992} C_VEL
LIN {X 0,Y 221.019,Z 292.577,A -85,B 0,C 180,E1 -20356.627,E2 -20356.627} C_VEL
LIN {X 0,Y 220.894,Z 292.577,A -85,B 0,C 180,E1 -20360.484,E2 -20360.484} C_VEL
LIN {X 0,Y 220.868,Z 292.598,A -85,B 0,C 180,E1 -20364.432,E2 -20364.432} C_VEL
LIN {X 0,Y 220.827,Z 292.587,A -85,B 0,C 180,E1 -20368.512,E2 -20368.512} C_VEL
LIN {X 0,Y 220.822,Z 292.602,A -85,B 0,C 180,E1 -20372.752,E2 -20372.752} C_VEL
LIN {X 0,Y 220.837,Z 292.593,A -85,B 0,C 180,E1 -20377.285,E2 -20377.285} C_VEL
LIN {X 0,Y 220.796,Z 292.594,A -85,B 0,C 180,E1 -20381.943,E2 -20381.943} C_VEL
LIN {X 0,Y 220.864,Z 292.597,A -85,B 0,C 180,E1 -20387.04,E2 -20387.04} C_VEL
LIN {X 0,Y 220.852,Z 292.593,A -85,B 0,C 180,E1 -20390.471,E2 -20390.471} C_VEL
LIN {X 0,Y 220.811,Z 292.595,A -85,B 0,C 180,E1 -20395.045,E2 -20395.045} C_VEL
LIN {X 0,Y 220.863,Z 292.595,A -85,B 0,C 180,E1 -20399.393,E2 -20399.393} C_VEL
LIN {X 0,Y 220.89,Z 292.596,A -85,B 0,C 180,E1 -20403.548,E2 -20403.548} C_VEL
LIN {X 0,Y 220.871,Z 292.6,A -85,B 0,C 180,E1 -20407.551,E2 -20407.551} C_VEL
LIN {X 0,Y 220.977,Z 292.578,A -85,B 0,C 180,E1 -20412.569,E2 -20412.569} C_VEL
LIN {X 0,Y 221.02,Z 292.712,A -85,B 0,C 180,E1 -20416.348,E2 -20416.348} C_VEL
LIN {X 0,Y 222.052,Z 295.504,A -85,B 0,C 180,E1 -20416.743,E2 -20416.743} C_VEL
LIN {X 0,Y 223.799,Z 297.756,A -85,B 0,C 180,E1 -20417.266,E2 -20417.266} C_VEL
LIN {X 0,Y 225.887,Z 301.14,A -85,B 0,C 180,E1 -20417.958,E2 -20417.958} C_VEL
LIN {X 0,Y 232.025,Z 311.542,A -85,B 0,C 180,E1 -20420.024,E2 -20420.024} C_VEL
LIN {X 0,Y 238.774,Z 326.681,A -85,B 0,C 180,E1 -20422.815,E2 -20422.815} C_VEL
LIN {X 0,Y 242.191,Z 339.543,A -85,B 0,C 180,E1 -20425.005,E2 -20425.005} C_VEL
LIN {X 0,Y 244.61,Z 349.841,A -85,B 0,C 180,E1 -20426.911,E2 -20426.911} C_VEL
LIN {X 0,Y 245.072,Z 353.353,A -85,B 0,C 180,E1 -20427.533,E2 -20427.533} C_VEL
LIN {X 0,Y 241.778,Z 366.29,A -85,B 0,C 180,E1 -20429.374,E2 -20429.374} C_VEL
LIN {X 0,Y 238.374,Z 378.325,A -85,B 0,C 180,E1 -20431.486,E2 -20431.486} C_VEL
LIN {X 0,Y 234.95,Z 389.414,A -85,B 0,C 180,E1 -20433.858,E2 -20433.858} C_VEL
LIN {X 0,Y 231.522,Z 399.716,A -85,B 0,C 180,E1 -20436.537,E2 -20436.537} C_VEL
LIN {X 0,Y 228.537,Z 408.277,A -85,B 0,C 180,E1 -20439.24,E2 -20439.24} C_VEL
LIN {X 0,Y 225.503,Z 416.94,A -85,B 0,C 180,E1 -20442.6,E2 -20442.6} C_VEL
LIN {X 0,Y 223.512,Z 423.003,A -85,B 0,C 180,E1 -20445.501,E2 -20445.501} C_VEL
LIN {X 0,Y 221.797,Z 428.095,A -85,B 0,C 180,E1 -20448.472,E2 -20448.472} C_VEL
LIN {X 0,Y 220.27,Z 433.171,A -85,B 0,C 180,E1 -20452.296,E2 -20452.296} C_VEL
LIN {X 0,Y 219.221,Z 436.835,A -85,B 0,C 180,E1 -20456.155,E2 -20456.155} C_VEL
LIN {X 0,Y 218.693,Z 439.07,A -85,B 0,C 180,E1 -20459.815,E2 -20459.815} C_VEL
LIN {X 0,Y 218.601,Z 440.159,A -85,B 0,C 180,E1 -20463.295,E2 -20463.295} C_VEL
LIN {X 0,Y 218.809,Z 440.281,A -85,B 0,C 180,E1 -20466.588,E2 -20466.588} C_VEL
LIN {X 0,Y 219.386,Z 439.473,A -85,B 0,C 180,E1 -20469.842,E2 -20469.842} C_VEL
LIN {X 0,Y 220.236,Z 438.035,A -85,B 0,C 180,E1 -20472.784,E2 -20472.784} C_VEL
LIN {X 0,Y 221.917,Z 434.843,A -85,B 0,C 180,E1 -20476.75,E2 -20476.75} C_VEL
LIN {X 0,Y 224.065,Z 430.818,A -85,B 0,C 180,E1 -20480.181,E2 -20480.181} C_VEL
LIN {X 0,Y 226.764,Z 425.414,A -85,B 0,C 180,E1 -20483.686,E2 -20483.686} C_VEL
LIN {X 0,Y 229.697,Z 419.74,A -85,B 0,C 180,E1 -20486.585,E2 -20486.585} C_VEL
LIN {X 0,Y 233.36,Z 412.254,A -85,B 0,C 180,E1 -20489.676,E2 -20489.676} C_VEL
LIN {X 0,Y 237.535,Z 403.468,A -85,B 0,C 180,E1 -20492.572,E2 -20492.572} C_VEL
LIN {X 0,Y 241.925,Z 393.589,A -85,B 0,C 180,E1 -20495.2,E2 -20495.2} C_VEL
LIN {X 0,Y 246.792,Z 381.688,A -85,B 0,C 180,E1 -20497.743,E2 -20497.743} C_VEL
LIN {X 0,Y 250.968,Z 370.224,A -85,B 0,C 180,E1 -20499.735,E2 -20499.735} C_VEL
LIN {X 0,Y 253.594,Z 361.936,A -85,B 0,C 180,E1 -20500.956,E2 -20500.956} C_VEL
LIN {X 0,Y 252.133,Z 351.61,A -85,B 0,C 180,E1 -20503.401,E2 -20503.401} C_VEL
LIN {X 0,Y 249.723,Z 342.283,A -85,B 0,C 180,E1 -20505.746,E2 -20505.746} C_VEL
LIN {X 0,Y 247.255,Z 335.244,A -85,B 0,C 180,E1 -20507.693,E2 -20507.693} C_VEL
LIN {X 0,Y 244.77,Z 329.607,A -85,B 0,C 180,E1 -20509.421,E2 -20509.421} C_VEL
LIN {X 0,Y 240.1,Z 320.915,A -85,B 0,C 180,E1 -20512.498,E2 -20512.498} C_VEL
LIN {X 0,Y 237.588,Z 316.841,A -85,B 0,C 180,E1 -20514.191,E2 -20514.191} C_VEL
LIN {X 0,Y 235.342,Z 313.494,A -85,B 0,C 180,E1 -20515.72,E2 -20515.72} C_VEL
LIN {X 0,Y 234.287,Z 312.214,A -85,B 0,C 180,E1 -20516.455,E2 -20516.455} C_VEL
LIN {X 0,Y 232.088,Z 309.29,A -85,B 0,C 180,E1 -20518.056,E2 -20518.056} C_VEL
LIN {X 0,Y 231.176,Z 307.6,A -85,B 0,C 180,E1 -20518.84,E2 -20518.84} C_VEL
LIN {X 0,Y 228.642,Z 305.104,A -85,B 0,C 180,E1 -20520.882,E2 -20520.882} C_VEL
LIN {X 0,Y 227.306,Z 302.68,A -85,B 0,C 180,E1 -20522.217,E2 -20522.217} C_VEL
LIN {X 0,Y 224.247,Z 301.143,A -85,B 0,C 180,E1 -20525.171,E2 -20525.171} C_VEL
LIN {X 0,Y 222.485,Z 298.75,A -85,B 0,C 180,E1 -20527.717,E2 -20527.717} C_VEL
LIN {X 0,Y 222.161,Z 297.726,A -85,B 0,C 180,E1 -20528.53,E2 -20528.53} C_VEL
LIN {X 0,Y 222.1,Z 298.345,A -85,B 0,C 180,E1 -20532.799,E2 -20532.799} C_VEL
LIN {X 0,Y 222.179,Z 299.165,A -85,B 0,C 180,E1 -20536.542,E2 -20536.542} C_VEL
LIN {X 0,Y 222.3,Z 300.297,A -85,B 0,C 180,E1 -20540.352,E2 -20540.352} C_VEL
LIN {X 0,Y 222.593,Z 302.187,A -85,B 0,C 180,E1 -20544.981,E2 -20544.981} C_VEL
LIN {X 0,Y 223.913,Z 305.549,A -85,B 0,C 180,E1 -20546.995,E2 -20546.995} C_VEL
LIN {X 0,Y 226.873,Z 309.533,A -85,B 0,C 180,E1 -20550.131,E2 -20550.131} C_VEL
LIN {X 0,Y 227.939,Z 310.589,A -85,B 0,C 180,E1 -20551.046,E2 -20551.046} C_VEL
LIN {X 0,Y 229.505,Z 314.23,A -85,B 0,C 180,E1 -20552.536,E2 -20552.536} C_VEL
LIN {X 0,Y 232.287,Z 317.865,A -85,B 0,C 180,E1 -20554.633,E2 -20554.633} C_VEL
LIN {X 0,Y 234.292,Z 322.098,A -85,B 0,C 180,E1 -20556.17,E2 -20556.17} C_VEL
LIN {X 0,Y 235.992,Z 324.645,A -85,B 0,C 180,E1 -20557.299,E2 -20557.299} C_VEL
LIN {X 0,Y 238.102,Z 329.021,A -85,B 0,C 180,E1 -20558.78,E2 -20558.78} C_VEL
LIN {X 0,Y 239.193,Z 330.937,A -85,B 0,C 180,E1 -20559.451,E2 -20559.451} C_VEL
LIN {X 0,Y 242.025,Z 337.092,A -85,B 0,C 180,E1 -20561.346,E2 -20561.346} C_VEL
LIN {X 0,Y 244.335,Z 343.384,A -85,B 0,C 180,E1 -20562.988,E2 -20562.988} C_VEL
LIN {X 0,Y 246.451,Z 353.274,A -85,B 0,C 180,E1 -20565.097,E2 -20565.097} C_VEL
LIN {X 0,Y 246.688,Z 358.034,A -85,B 0,C 180,E1 -20565.907,E2 -20565.907} C_VEL
LIN {X 0,Y 245.781,Z 364.882,A -85,B 0,C 180,E1 -20566.814,E2 -20566.814} C_VEL
LIN {X 0,Y 243.744,Z 373.543,A -85,B 0,C 180,E1 -20567.904,E2 -20567.904} C_VEL
LIN {X 0,Y 242.855,Z 378.515,A -85,B 0,C 180,E1 -20568.678,E2 -20568.678} C_VEL
LIN {X 0,Y 242.719,Z 380.042,A -85,B 0,C 180,E1 -20568.973,E2 -20568.973} C_VEL
LIN {X 0,Y 241.807,Z 390.843,A -85,B 0,C 180,E1 -20571.141,E2 -20571.141} C_VEL
LIN {X 0,Y 240.751,Z 397.253,A -85,B 0,C 180,E1 -20572.457,E2 -20572.457} C_VEL
LIN {X 0,Y 236.14,Z 408.397,A -85,B 0,C 180,E1 -20574.526,E2 -20574.526} C_VEL
LIN {X 0,Y 231.552,Z 418.761,A -85,B 0,C 180,E1 -20576.886,E2 -20576.886} C_VEL
LIN {X 0,Y 226.803,Z 429.017,A -85,B 0,C 180,E1 -20579.767,E2 -20579.767} C_VEL
LIN {X 0,Y 222.859,Z 437.663,A -85,B 0,C 180,E1 -20582.791,E2 -20582.791} C_VEL
LIN {X 0,Y 218.916,Z 445.865,A -85,B 0,C 180,E1 -20586.342,E2 -20586.342} C_VEL
LIN {X 0,Y 215.89,Z 452.514,A -85,B 0,C 180,E1 -20590.014,E2 -20590.014} C_VEL
LIN {X 0,Y 213.704,Z 457.797,A -85,B 0,C 180,E1 -20593.769,E2 -20593.769} C_VEL
LIN {X 0,Y 212.626,Z 460.917,A -85,B 0,C 180,E1 -20596.623,E2 -20596.623} C_VEL
LIN {X 0,Y 211.838,Z 464.018,A -85,B 0,C 180,E1 -20600.453,E2 -20600.453} C_VEL
LIN {X 0,Y 211.707,Z 465.964,A -85,B 0,C 180,E1 -20604.286,E2 -20604.286} C_VEL
LIN {X 0,Y 211.755,Z 466.743,A -85,B 0,C 180,E1 -20608.099,E2 -20608.099} C_VEL
LIN {X 0,Y 211.786,Z 466.661,A -85,B 0,C 180,E1 -20610.001,E2 -20610.001} C_VEL
LIN {X 0,Y 211.741,Z 465.59,A -85,B 0,C 180,E1 -20613.808,E2 -20613.808} C_VEL
LIN {X 0,Y 211.809,Z 464.606,A -85,B 0,C 180,E1 -20615.714,E2 -20615.714} C_VEL
LIN {X 0,Y 211.88,Z 461.681,A -85,B 0,C 180,E1 -20619.548,E2 -20619.548} C_VEL
LIN {X 0,Y 212.646,Z 457.474,A -85,B 0,C 180,E1 -20623.378,E2 -20623.378} C_VEL
LIN {X 0,Y 214.127,Z 451.868,A -85,B 0,C 180,E1 -20627.182,E2 -20627.182} C_VEL
LIN {X 0,Y 216.388,Z 444.719,A -85,B 0,C 180,E1 -20630.934,E2 -20630.934} C_VEL
LIN {X 0,Y 219.066,Z 437.069,A -85,B 0,C 180,E1 -20634.146,E2 -20634.146} C_VEL
LIN {X 0,Y 222.304,Z 427.867,A -85,B 0,C 180,E1 -20637.279,E2 -20637.279} C_VEL
LIN {X 0,Y 225.586,Z 418.429,A -85,B 0,C 180,E1 -20639.9,E2 -20639.9} C_VEL
LIN {X 0,Y 229.74,Z 406.35,A -85,B 0,C 180,E1 -20642.628,E2 -20642.628} C_VEL
LIN {X 0,Y 233.271,Z 395.22,A -85,B 0,C 180,E1 -20644.659,E2 -20644.659} C_VEL
LIN {X 0,Y 234.29,Z 391.257,A -85,B 0,C 180,E1 -20645.313,E2 -20645.313} C_VEL
LIN {X 0,Y 234.061,Z 378.824,A -85,B 0,C 180,E1 -20647.579,E2 -20647.579} C_VEL
LIN {X 0,Y 232.985,Z 365.73,A -85,B 0,C 180,E1 -20649.759,E2 -20649.759} C_VEL
LIN {X 0,Y 230.946,Z 352.574,A -85,B 0,C 180,E1 -20651.791,E2 -20651.791} C_VEL
LIN {X 0,Y 227.892,Z 338.487,A -85,B 0,C 180,E1 -20653.826,E2 -20653.826} C_VEL
LIN {X 0,Y 224.557,Z 326.977,A -85,B 0,C 180,E1 -20655.471,E2 -20655.471} C_VEL
LIN {X 0,Y 220.973,Z 318.657,A -85,B 0,C 180,E1 -20656.795,E2 -20656.795} C_VEL
LIN {X 0,Y 218.519,Z 313.909,A -85,B 0,C 180,E1 -20657.602,E2 -20657.602} C_VEL
LIN {X 0,Y 216.847,Z 310.717,A -85,B 0,C 180,E1 -20658.159,E2 -20658.159} C_VEL
LIN {X 0,Y 216.526,Z 309.312,A -85,B 0,C 180,E1 -20658.371,E2 -20658.371} C_VEL
LIN {X 0,Y 215.89,Z 306.306,A -85,B 0,C 180,E1 -20661.79,E2 -20661.79} C_VEL
LIN {X 0,Y 215.254,Z 302.562,A -85,B 0,C 180,E1 -20666.284,E2 -20666.284} C_VEL
LIN {X 0,Y 214.735,Z 299.239,A -85,B 0,C 180,E1 -20670.596,E2 -20670.596} C_VEL
LIN {X 0,Y 214.305,Z 296.259,A -85,B 0,C 180,E1 -20674.763,E2 -20674.763} C_VEL
LIN {X 0,Y 213.861,Z 293.47,A -85,B 0,C 180,E1 -20679.311,E2 -20679.311} C_VEL
LIN {X 0,Y 213.951,Z 293.462,A -85,B 0,C 180,E1 -20682.802,E2 -20682.802} C_VEL
LIN {X 0,Y 213.96,Z 293.462,A -85,B 0,C 180,E1 -20686.705,E2 -20686.705} C_VEL
LIN {X 0,Y 214.143,Z 293.44,A -85,B 0,C 180,E1 -20690.553,E2 -20690.553} C_VEL
LIN {X 0,Y 214.097,Z 293.444,A -85,B 0,C 180,E1 -20694.346,E2 -20694.346} C_VEL
LIN {X 0,Y 214.449,Z 293.398,A -85,B 0,C 180,E1 -20698.12,E2 -20698.12} C_VEL
LIN {X 0,Y 214.556,Z 293.384,A -85,B 0,C 180,E1 -20699.998,E2 -20699.998} C_VEL
LIN {X 0,Y 214.45,Z 293.395,A -85,B 0,C 180,E1 -20701.876,E2 -20701.876} C_VEL
LIN {X 0,Y 214.252,Z 293.419,A -85,B 0,C 180,E1 -20707.537,E2 -20707.537} C_VEL
LIN {X 0,Y 214.03,Z 293.434,A -85,B 0,C 180,E1 -20711.361,E2 -20711.361} C_VEL
LIN {X 0,Y 213.937,Z 293.458,A -85,B 0,C 180,E1 -20715.234,E2 -20715.234} C_VEL
LIN {X 0,Y 213.842,Z 293.459,A -85,B 0,C 180,E1 -20719.185,E2 -20719.185} C_VEL
LIN {X 0,Y 213.849,Z 293.47,A -85,B 0,C 180,E1 -20723.224,E2 -20723.224} C_VEL
LIN {X 0,Y 213.83,Z 293.459,A -85,B 0,C 180,E1 -20727.447,E2 -20727.447} C_VEL
LIN {X 0,Y 213.77,Z 293.482,A -85,B 0,C 180,E1 -20731.734,E2 -20731.734} C_VEL
LIN {X 0,Y 213.751,Z 293.469,A -85,B 0,C 180,E1 -20736.284,E2 -20736.284} C_VEL
LIN {X 0,Y 213.73,Z 293.482,A -85,B 0,C 180,E1 -20741.118,E2 -20741.118} C_VEL
LIN {X 0,Y 213.808,Z 293.477,A -85,B 0,C 180,E1 -20746.346,E2 -20746.346} C_VEL
LIN {X 0,Y 213.791,Z 293.467,A -85,B 0,C 180,E1 -20749.116,E2 -20749.116} C_VEL
LIN {X 0,Y 213.75,Z 293.479,A -85,B 0,C 180,E1 -20753.711,E2 -20753.711} C_VEL
LIN {X 0,Y 213.791,Z 293.48,A -85,B 0,C 180,E1 -20758.722,E2 -20758.722} C_VEL
LIN {X 0,Y 213.82,Z 293.479,A -85,B 0,C 180,E1 -20762.601,E2 -20762.601} C_VEL
LIN {X 0,Y 213.846,Z 293.476,A -85,B 0,C 180,E1 -20766.951,E2 -20766.951} C_VEL
LIN {X 0,Y 213.925,Z 293.457,A -85,B 0,C 180,E1 -20772.303,E2 -20772.303} C_VEL
LIN {X 0,Y 213.952,Z 293.547,A -85,B 0,C 180,E1 -20774.733,E2 -20774.733} C_VEL
LIN {X 0,Y 214.889,Z 296.213,A -85,B 0,C 180,E1 -20775.121,E2 -20775.121} C_VEL
LIN {X 0,Y 216.78,Z 298.711,A -85,B 0,C 180,E1 -20775.731,E2 -20775.731} C_VEL
LIN {X 0,Y 218.856,Z 302.046,A -85,B 0,C 180,E1 -20776.461,E2 -20776.461} C_VEL
LIN {X 0,Y 226.135,Z 314.398,A -85,B 0,C 180,E1 -20779.11,E2 -20779.11} C_VEL
LIN {X 0,Y 230.046,Z 322.954,A -85,B 0,C 180,E1 -20780.779,E2 -20780.779} C_VEL
LIN {X 0,Y 233.551,Z 331.423,A -85,B 0,C 180,E1 -20782.449,E2 -20782.449} C_VEL
LIN {X 0,Y 236.784,Z 344.953,A -85,B 0,C 180,E1 -20784.89,E2 -20784.89} C_VEL
LIN {X 0,Y 238.706,Z 353.864,A -85,B 0,C 180,E1 -20786.623,E2 -20786.623} C_VEL
LIN {X 0,Y 238.718,Z 355.065,A -85,B 0,C 180,E1 -20786.834,E2 -20786.834} C_VEL
LIN {X 0,Y 235.289,Z 367.833,A -85,B 0,C 180,E1 -20788.715,E2 -20788.715} C_VEL
LIN {X 0,Y 231.936,Z 379.304,A -85,B 0,C 180,E1 -20790.801,E2 -20790.801} C_VEL
LIN {X 0,Y 228.584,Z 389.69,A -85,B 0,C 180,E1 -20793.083,E2 -20793.083} C_VEL
LIN {X 0,Y 225.007,Z 400.018,A -85,B 0,C 180,E1 -20795.825,E2 -20795.825} C_VEL
LIN {X 0,Y 221.839,Z 408.758,A -85,B 0,C 180,E1 -20798.654,E2 -20798.654} C_VEL
LIN {X 0,Y 218.732,Z 417.29,A -85,B 0,C 180,E1 -20802.054,E2 -20802.054} C_VEL
LIN {X 0,Y 216.644,Z 423.371,A -85,B 0,C 180,E1 -20805.04,E2 -20805.04} C_VEL
LIN {X 0,Y 214.738,Z 428.877,A -85,B 0,C 180,E1 -20808.364,E2 -20808.364} C_VEL
LIN {X 0,Y 213.062,Z 434.127,A -85,B 0,C 180,E1 -20812.549,E2 -20812.549} C_VEL
LIN {X 0,Y 212.043,Z 437.625,A -85,B 0,C 180,E1 -20816.511,E2 -20816.511} C_VEL
LIN {X 0,Y 211.591,Z 439.71,A -85,B 0,C 180,E1 -20820.283,E2 -20820.283} C_VEL
LIN {X 0,Y 211.544,Z 440.728,A -85,B 0,C 180,E1 -20824.385,E2 -20824.385} C_VEL
LIN {X 0,Y 211.83,Z 440.699,A -85,B 0,C 180,E1 -20827.23,E2 -20827.23} C_VEL
LIN {X 0,Y 212.676,Z 439.51,A -85,B 0,C 180,E1 -20831.367,E2 -20831.367} C_VEL
LIN {X 0,Y 213.483,Z 438.198,A -85,B 0,C 180,E1 -20833.734,E2 -20833.734} C_VEL
LIN {X 0,Y 214.727,Z 435.993,A -85,B 0,C 180,E1 -20836.585,E2 -20836.585} C_VEL
LIN {X 0,Y 216.412,Z 433.048,A -85,B 0,C 180,E1 -20839.499,E2 -20839.499} C_VEL
LIN {X 0,Y 219.239,Z 427.945,A -85,B 0,C 180,E1 -20843.262,E2 -20843.262} C_VEL
LIN {X 0,Y 222.51,Z 421.884,A -85,B 0,C 180,E1 -20846.673,E2 -20846.673} C_VEL
LIN {X 0,Y 226.824,Z 413.659,A -85,B 0,C 180,E1 -20850.283,E2 -20850.283} C_VEL
LIN {X 0,Y 230.924,Z 405.512,A -85,B 0,C 180,E1 -20853.105,E2 -20853.105} C_VEL
LIN {X 0,Y 235.565,Z 395.723,A -85,B 0,C 180,E1 -20855.855,E2 -20855.855} C_VEL
LIN {X 0,Y 239.787,Z 386.168,A -85,B 0,C 180,E1 -20858.034,E2 -20858.034} C_VEL
LIN {X 0,Y 244.181,Z 374.984,A -85,B 0,C 180,E1 -20860.155,E2 -20860.155} C_VEL
LIN {X 0,Y 247.955,Z 364.319,A -85,B 0,C 180,E1 -20861.835,E2 -20861.835} C_VEL
LIN {X 0,Y 246.848,Z 355.248,A -85,B 0,C 180,E1 -20864.098,E2 -20864.098} C_VEL
LIN {X 0,Y 244.626,Z 345.539,A -85,B 0,C 180,E1 -20866.715,E2 -20866.715} C_VEL
LIN {X 0,Y 241.639,Z 337.006,A -85,B 0,C 180,E1 -20869.283,E2 -20869.283} C_VEL
LIN {X 0,Y 238.073,Z 329.564,A -85,B 0,C 180,E1 -20871.941,E2 -20871.941} C_VEL
LIN {X 0,Y 236.478,Z 326.413,A -85,B 0,C 180,E1 -20873.175,E2 -20873.175} C_VEL
LIN {X 0,Y 234.34,Z 322.781,A -85,B 0,C 180,E1 -20874.749,E2 -20874.749} C_VEL
LIN {X 0,Y 231.864,Z 318.789,A -85,B 0,C 180,E1 -20876.717,E2 -20876.717} C_VEL
LIN {X 0,Y 229.607,Z 315.776,A -85,B 0,C 180,E1 -20878.491,E2 -20878.491} C_VEL
LIN {X 0,Y 228.907,Z 314.18,A -85,B 0,C 180,E1 -20879.218,E2 -20879.218} C_VEL
LIN {X 0,Y 226.375,Z 311.458,A -85,B 0,C 180,E1 -20881.447,E2 -20881.447} C_VEL
LIN {X 0,Y 225.458,Z 309.606,A -85,B 0,C 180,E1 -20882.515,E2 -20882.515} C_VEL
LIN {X 0,Y 222.176,Z 307.491,A -85,B 0,C 180,E1 -20886.13,E2 -20886.13} C_VEL
LIN {X 0,Y 220.772,Z 304.734,A -85,B 0,C 180,E1 -20888.7,E2 -20888.7} C_VEL
LIN {X 0,Y 218.497,Z 304.936,A -85,B 0,C 180,E1 -20895.219,E2 -20895.219} C_VEL
LIN {X 0,Y 218.959,Z 306.464,A -85,B 0,C 180,E1 -20899.942,E2 -20899.942} C_VEL
LIN {X 0,Y 221.084,Z 309.028,A -85,B 0,C 180,E1 -20904.536,E2 -20904.536} C_VEL
LIN {X 0,Y 222.442,Z 312.612,A -85,B 0,C 180,E1 -20906.814,E2 -20906.814} C_VEL
LIN {X 0,Y 225.789,Z 317.235,A -85,B 0,C 180,E1 -20910.516,E2 -20910.516} C_VEL
LIN {X 0,Y 227.399,Z 320.997,A -85,B 0,C 180,E1 -20912.219,E2 -20912.219} C_VEL
LIN {X 0,Y 229.588,Z 324.034,A -85,B 0,C 180,E1 -20914.009,E2 -20914.009} C_VEL
LIN {X 0,Y 231.431,Z 328.215,A -85,B 0,C 180,E1 -20915.641,E2 -20915.641} C_VEL
LIN {X 0,Y 232.895,Z 330.658,A -85,B 0,C 180,E1 -20916.703,E2 -20916.703} C_VEL
LIN {X 0,Y 235.001,Z 335.156,A -85,B 0,C 180,E1 -20918.358,E2 -20918.358} C_VEL
LIN {X 0,Y 238.334,Z 342.99,A -85,B 0,C 180,E1 -20920.873,E2 -20920.873} C_VEL
LIN {X 0,Y 240.055,Z 348.365,A -85,B 0,C 180,E1 -20922.329,E2 -20922.329} C_VEL
LIN {X 0,Y 241.705,Z 357.954,A -85,B 0,C 180,E1 -20924.462,E2 -20924.462} C_VEL
LIN {X 0,Y 242.769,Z 370.101,A -85,B 0,C 180,E1 -20926.97,E2 -20926.97} C_VEL
LIN {X 0,Y 242.719,Z 380.042,A -85,B 0,C 180,E1 -20928.973,E2 -20928.973} C_VEL
LIN {X 0,Y 241.864,Z 384.822,A -85,B 0,C 180,E1 -20929.795,E2 -20929.795} C_VEL
LIN {X 0,Y 240.063,Z 389.68,A -85,B 0,C 180,E1 -20930.492,E2 -20930.492} C_VEL
LIN {X 0,Y 235.075,Z 399.292,A -85,B 0,C 180,E1 -20931.795,E2 -20931.795} C_VEL
LIN {X 0,Y 231.935,Z 405.411,A -85,B 0,C 180,E1 -20932.832,E2 -20932.832} C_VEL
LIN {X 0,Y 227.174,Z 415.787,A -85,B 0,C 180,E1 -20935.089,E2 -20935.089} C_VEL
LIN {X 0,Y 222.015,Z 426.438,A -85,B 0,C 180,E1 -20937.981,E2 -20937.981} C_VEL
LIN {X 0,Y 217.571,Z 435.408,A -85,B 0,C 180,E1 -20941.02,E2 -20941.02} C_VEL
LIN {X 0,Y 213.832,Z 442.933,A -85,B 0,C 180,E1 -20944.185,E2 -20944.185} C_VEL
LIN {X 0,Y 210.644,Z 449.23,A -85,B 0,C 180,E1 -20947.439,E2 -20947.439} C_VEL
LIN {X 0,Y 207.75,Z 455.163,A -85,B 0,C 180,E1 -20951.305,E2 -20951.305} C_VEL
LIN {X 0,Y 206.378,Z 458.664,A -85,B 0,C 180,E1 -20954.192,E2 -20954.192} C_VEL
LIN {X 0,Y 205.123,Z 462.29,A -85,B 0,C 180,E1 -20958.138,E2 -20958.138} C_VEL
LIN {X 0,Y 204.635,Z 464.754,A -85,B 0,C 180,E1 -20962.105,E2 -20962.105} C_VEL
LIN {X 0,Y 204.597,Z 466.069,A -85,B 0,C 180,E1 -20966.062,E2 -20966.062} C_VEL
LIN {X 0,Y 204.687,Z 466.296,A -85,B 0,C 180,E1 -20968.034,E2 -20968.034} C_VEL
LIN {X 0,Y 204.719,Z 466.206,A -85,B 0,C 180,E1 -20970.001,E2 -20970.001} C_VEL
LIN {X 0,Y 204.67,Z 465.079,A -85,B 0,C 180,E1 -20973.939,E2 -20973.939} C_VEL
LIN {X 0,Y 204.709,Z 464.063,A -85,B 0,C 180,E1 -20975.913,E2 -20975.913} C_VEL
LIN {X 0,Y 204.834,Z 461.08,A -85,B 0,C 180,E1 -20979.879,E2 -20979.879} C_VEL
LIN {X 0,Y 205.69,Z 456.811,A -85,B 0,C 180,E1 -20983.839,E2 -20983.839} C_VEL
LIN {X 0,Y 207.269,Z 451.136,A -85,B 0,C 180,E1 -20987.77,E2 -20987.77} C_VEL
LIN {X 0,Y 209.667,Z 443.912,A -85,B 0,C 180,E1 -20991.638,E2 -20991.638} C_VEL
LIN {X 0,Y 212.541,Z 436.187,A -85,B 0,C 180,E1 -20994.937,E2 -20994.937} C_VEL
LIN {X 0,Y 215.745,Z 427.305,A -85,B 0,C 180,E1 -20998.034,E2 -20998.034} C_VEL
LIN {X 0,Y 219.387,Z 417.404,A -85,B 0,C 180,E1 -21000.836,E2 -21000.836} C_VEL
LIN {X 0,Y 223.656,Z 405.154,A -85,B 0,C 180,E1 -21003.632,E2 -21003.632} C_VEL
LIN {X 0,Y 227.736,Z 392.706,A -85,B 0,C 180,E1 -21005.899,E2 -21005.899} C_VEL
LIN {X 0,Y 227.66,Z 379.697,A -85,B 0,C 180,E1 -21008.386,E2 -21008.386} C_VEL
LIN {X 0,Y 226.539,Z 365.551,A -85,B 0,C 180,E1 -21010.835,E2 -21010.835} C_VEL
LIN {X 0,Y 224.258,Z 350.61,A -85,B 0,C 180,E1 -21013.226,E2 -21013.226} C_VEL
LIN {X 0,Y 220.806,Z 335.682,A -85,B 0,C 180,E1 -21015.508,E2 -21015.508} C_VEL
LIN {X 0,Y 217.884,Z 326.868,A -85,B 0,C 180,E1 -21016.887,E2 -21016.887} C_VEL
LIN {X 0,Y 213.797,Z 318.3,A -85,B 0,C 180,E1 -21018.43,E2 -21018.43} C_VEL
LIN {X 0,Y 211.975,Z 314.522,A -85,B 0,C 180,E1 -21019.093,E2 -21019.093} C_VEL
LIN {X 0,Y 209.678,Z 310.691,A -85,B 0,C 180,E1 -21019.894,E2 -21019.894} C_VEL
LIN {X 0,Y 209.142,Z 308.813,A -85,B 0,C 180,E1 -21020.163,E2 -21020.163} C_VEL
LIN {X 0,Y 208.4,Z 304.804,A -85,B 0,C 180,E1 -21025.017,E2 -21025.017} C_VEL
LIN {X 0,Y 207.866,Z 301.34,A -85,B 0,C 180,E1 -21029.524,E2 -21029.524} C_VEL
LIN {X 0,Y 207.422,Z 298.257,A -85,B 0,C 180,E1 -21033.864,E2 -21033.864} C_VEL
LIN {X 0,Y 206.903,Z 294.893,A -85,B 0,C 180,E1 -21039.103,E2 -21039.103} C_VEL
LIN {X 0,Y 206.823,Z 294.347,A -85,B 0,C 180,E1 -21040.133,E2 -21040.133} C_VEL
LIN {X 0,Y 206.874,Z 294.344,A -85,B 0,C 180,E1 -21044.228,E2 -21044.228} C_VEL
LIN {X 0,Y 207.067,Z 294.32,A -85,B 0,C 180,E1 -21049.834,E2 -21049.834} C_VEL
LIN {X 0,Y 207.138,Z 294.312,A -85,B 0,C 180,E1 -21052.198,E2 -21052.198} C_VEL
LIN {X 0,Y 207.385,Z 294.278,A -85,B 0,C 180,E1 -21058.056,E2 -21058.056} C_VEL
LIN {X 0,Y 207.52,Z 294.26,A -85,B 0,C 180,E1 -21059.998,E2 -21059.998} C_VEL
LIN {X 0,Y 207.387,Z 294.274,A -85,B 0,C 180,E1 -21061.94,E2 -21061.94} C_VEL
LIN {X 0,Y 207.193,Z 294.299,A -85,B 0,C 180,E1 -21067.796,E2 -21067.796} C_VEL
LIN {X 0,Y 206.949,Z 294.313,A -85,B 0,C 180,E1 -21071.755,E2 -21071.755} C_VEL
LIN {X 0,Y 206.87,Z 294.339,A -85,B 0,C 180,E1 -21075.768,E2 -21075.768} C_VEL
LIN {X 0,Y 206.786,Z 294.333,A -85,B 0,C 180,E1 -21079.866,E2 -21079.866} C_VEL
LIN {X 0,Y 206.765,Z 294.356,A -85,B 0,C 180,E1 -21084.069,E2 -21084.069} C_VEL
LIN {X 0,Y 206.737,Z 294.34,A -85,B 0,C 180,E1 -21088.417,E2 -21088.417} C_VEL
LIN {X 0,Y 206.705,Z 294.36,A -85,B 0,C 180,E1 -21092.954,E2 -21092.954} C_VEL
LIN {X 0,Y 206.721,Z 294.344,A -85,B 0,C 180,E1 -21095.318,E2 -21095.318} C_VEL
LIN {X 0,Y 206.673,Z 294.364,A -85,B 0,C 180,E1 -21100.245,E2 -21100.245} C_VEL
LIN {X 0,Y 206.705,Z 294.361,A -85,B 0,C 180,E1 -21105.558,E2 -21105.558} C_VEL
LIN {X 0,Y 206.721,Z 294.347,A -85,B 0,C 180,E1 -21109.761,E2 -21109.761} C_VEL
LIN {X 0,Y 206.721,Z 294.36,A -85,B 0,C 180,E1 -21112.267,E2 -21112.267} C_VEL
LIN {X 0,Y 206.704,Z 294.362,A -85,B 0,C 180,E1 -21117.042,E2 -21117.042} C_VEL
LIN {X 0,Y 206.761,Z 294.359,A -85,B 0,C 180,E1 -21122.094,E2 -21122.094} C_VEL
LIN {X 0,Y 206.779,Z 294.356,A -85,B 0,C 180,E1 -21126.582,E2 -21126.582} C_VEL
LIN {X 0,Y 206.869,Z 294.336,A -85,B 0,C 180,E1 -21132.195,E2 -21132.195} C_VEL
LIN {X 0,Y 206.9,Z 294.332,A -85,B 0,C 180,E1 -21132.963,E2 -21132.963} C_VEL
LIN {X 0,Y 207.92,Z 297.216,A -85,B 0,C 180,E1 -21133.431,E2 -21133.431} C_VEL
LIN {X 0,Y 209.794,Z 299.626,A -85,B 0,C 180,E1 -21134.09,E2 -21134.09} C_VEL
LIN {X 0,Y 211.866,Z 302.932,A -85,B 0,C 180,E1 -21134.872,E2 -21134.872} C_VEL
LIN {X 0,Y 219.498,Z 315.796,A -85,B 0,C 180,E1 -21137.83,E2 -21137.83} C_VEL
LIN {X 0,Y 223.237,Z 323.329,A -85,B 0,C 180,E1 -21139.458,E2 -21139.458} C_VEL
LIN {X 0,Y 228.013,Z 335.499,A -85,B 0,C 180,E1 -21141.941,E2 -21141.941} C_VEL
LIN {X 0,Y 230.932,Z 348.546,A -85,B 0,C 180,E1 -21144.442,E2 -21144.442} C_VEL
LIN {X 0,Y 232.35,Z 355.514,A -85,B 0,C 180,E1 -21145.879,E2 -21145.879} C_VEL
LIN {X 0,Y 232.39,Z 356.655,A -85,B 0,C 180,E1 -21146.097,E2 -21146.097} C_VEL
LIN {X 0,Y 228.85,Z 369.232,A -85,B 0,C 180,E1 -21148.019,E2 -21148.019} C_VEL
LIN {X 0,Y 225.181,Z 381.146,A -85,B 0,C 180,E1 -21150.271,E2 -21150.271} C_VEL
LIN {X 0,Y 221.589,Z 391.819,A -85,B 0,C 180,E1 -21152.726,E2 -21152.726} C_VEL
LIN {X 0,Y 217.976,Z 401.877,A -85,B 0,C 180,E1 -21155.549,E2 -21155.549} C_VEL
LIN {X 0,Y 214.182,Z 411.724,A -85,B 0,C 180,E1 -21158.966,E2 -21158.966} C_VEL
LIN {X 0,Y 211.257,Z 419.775,A -85,B 0,C 180,E1 -21162.487,E2 -21162.487} C_VEL
LIN {X 0,Y 209.085,Z 425.525,A -85,B 0,C 180,E1 -21165.598,E2 -21165.598} C_VEL
LIN {X 0,Y 207.515,Z 429.967,A -85,B 0,C 180,E1 -21168.515,E2 -21168.515} C_VEL
LIN {X 0,Y 205.889,Z 435.018,A -85,B 0,C 180,E1 -21172.84,E2 -21172.84} C_VEL
LIN {X 0,Y 204.887,Z 438.343,A -85,B 0,C 180,E1 -21176.9,E2 -21176.9} C_VEL
LIN {X 0,Y 204.452,Z 440.424,A -85,B 0,C 180,E1 -21181.037,E2 -21181.037} C_VEL
LIN {X 0,Y 204.46,Z 441.157,A -85,B 0,C 180,E1 -21184.42,E2 -21184.42} C_VEL
LIN {X 0,Y 204.866,Z 441.041,A -85,B 0,C 180,E1 -21188.132,E2 -21188.132} C_VEL
LIN {X 0,Y 205.558,Z 440.187,A -85,B 0,C 180,E1 -21191.225,E2 -21191.225} C_VEL
LIN {X 0,Y 207.079,Z 437.857,A -85,B 0,C 180,E1 -21195.454,E2 -21195.454} C_VEL
LIN {X 0,Y 209.047,Z 434.646,A -85,B 0,C 180,E1 -21199.148,E2 -21199.148} C_VEL
LIN {X 0,Y 211.687,Z 430.249,A -85,B 0,C 180,E1 -21202.823,E2 -21202.823} C_VEL
LIN {X 0,Y 214.797,Z 424.965,A -85,B 0,C 180,E1 -21206.208,E2 -21206.208} C_VEL
LIN {X 0,Y 219.133,Z 417.305,A -85,B 0,C 180,E1 -21209.987,E2 -21209.987} C_VEL
LIN {X 0,Y 223.097,Z 409.956,A -85,B 0,C 180,E1 -21212.862,E2 -21212.862} C_VEL
LIN {X 0,Y 227.609,Z 401.2,A -85,B 0,C 180,E1 -21215.625,E2 -21215.625} C_VEL
LIN {X 0,Y 232.598,Z 390.75,A -85,B 0,C 180,E1 -21218.294,E2 -21218.294} C_VEL
LIN {X 0,Y 237.479,Z 379.509,A -85,B 0,C 180,E1 -21220.611,E2 -21220.611} C_VEL
LIN {X 0,Y 242.351,Z 366.855,A -85,B 0,C 180,E1 -21222.71,E2 -21222.71} C_VEL
LIN {X 0,Y 241.33,Z 357.411,A -85,B 0,C 180,E1 -21225.239,E2 -21225.239} C_VEL
LIN {X 0,Y 239.483,Z 348.758,A -85,B 0,C 180,E1 -21227.718,E2 -21227.718} C_VEL
LIN {X 0,Y 236.91,Z 340.954,A -85,B 0,C 180,E1 -21230.272,E2 -21230.272} C_VEL
LIN {X 0,Y 233.101,Z 332.444,A -85,B 0,C 180,E1 -21233.576,E2 -21233.576} C_VEL
LIN {X 0,Y 231.656,Z 329.66,A -85,B 0,C 180,E1 -21234.78,E2 -21234.78} C_VEL
LIN {X 0,Y 228.573,Z 324.661,A -85,B 0,C 180,E1 -21237.427,E2 -21237.427} C_VEL
LIN {X 0,Y 226.582,Z 321.29,A -85,B 0,C 180,E1 -21239.359,E2 -21239.359} C_VEL
LIN {X 0,Y 225.947,Z 320.323,A -85,B 0,C 180,E1 -21240.002,E2 -21240.002} C_VEL
LIN {X 0,Y 223.555,Z 316.93,A -85,B 0,C 180,E1 -21242.536,E2 -21242.536} C_VEL
LIN {X 0,Y 223.192,Z 316.198,A -85,B 0,C 180,E1 -21243.02,E2 -21243.02} C_VEL
LIN {X 0,Y 220.551,Z 314.434,A -85,B 0,C 180,E1 -21246.176,E2 -21246.176} C_VEL
LIN {X 0,Y 219.027,Z 311.64,A -85,B 0,C 180,E1 -21249.234,E2 -21249.234} C_VEL
LIN {X 0,Y 217.111,Z 312.064,A -85,B 0,C 180,E1 -21255.973,E2 -21255.973} C_VEL
LIN {X 0,Y 217.829,Z 313.865,A -85,B 0,C 180,E1 -21260.789,E2 -21260.789} C_VEL
LIN {X 0,Y 219.346,Z 315.781,A -85,B 0,C 180,E1 -21264.08,E2 -21264.08} C_VEL
LIN {X 0,Y 220.642,Z 319.506,A -85,B 0,C 180,E1 -21266.575,E2 -21266.575} C_VEL
LIN {X 0,Y 223.36,Z 323.58,A -85,B 0,C 180,E1 -21269.904,E2 -21269.904} C_VEL
LIN {X 0,Y 224.956,Z 327.491,A -85,B 0,C 180,E1 -21271.819,E2 -21271.819} C_VEL
LIN {X 0,Y 226.77,Z 330.369,A -85,B 0,C 180,E1 -21273.47,E2 -21273.47} C_VEL
LIN {X 0,Y 228.853,Z 335.03,A -85,B 0,C 180,E1 -21275.487,E2 -21275.487} C_VEL
LIN {X 0,Y 229.584,Z 336.55,A -85,B 0,C 180,E1 -21276.108,E2 -21276.108} C_VEL
LIN {X 0,Y 232.123,Z 342.628,A -85,B 0,C 180,E1 -21278.366,E2 -21278.366} C_VEL
LIN {X 0,Y 234.57,Z 348.928,A -85,B 0,C 180,E1 -21280.467,E2 -21280.467} C_VEL
LIN {X 0,Y 235.946,Z 355.062,A -85,B 0,C 180,E1 -21282.083,E2 -21282.083} C_VEL
LIN {X 0,Y 237.012,Z 364.481,A -85,B 0,C 180,E1 -21284.238,E2 -21284.238} C_VEL
LIN {X 0,Y 237.402,Z 375.826,A -85,B 0,C 180,E1 -21286.7,E2 -21286.7} C_VEL
LIN {X 0,Y 236.813,Z 386.121,A -85,B 0,C 180,E1 -21288.88,E2 -21288.88} C_VEL
LIN {X 0,Y 235.264,Z 396.733,A -85,B 0,C 180,E1 -21291.148,E2 -21291.148} C_VEL
LIN {X 0,Y 234.447,Z 399.497,A -85,B 0,C 180,E1 -21291.719,E2 -21291.719} C_VEL
LIN {X 0,Y 231.935,Z 405.411,A -85,B 0,C 180,E1 -21292.832,E2 -21292.832} C_VEL
LIN {X 0,Y 229.453,Z 409.787,A -85,B 0,C 180,E1 -21293.618,E2 -21293.618} C_VEL
LIN {X 0,Y 223.907,Z 416.66,A -85,B 0,C 180,E1 -21294.757,E2 -21294.757} C_VEL
LIN {X 0,Y 218.352,Z 423.153,A -85,B 0,C 180,E1 -21296.045,E2 -21296.045} C_VEL
LIN {X 0,Y 215.881,Z 426.836,A -85,B 0,C 180,E1 -21297.062,E2 -21297.062} C_VEL
LIN {X 0,Y 211.345,Z 435.445,A -85,B 0,C 180,E1 -21300.081,E2 -21300.081} C_VEL
LIN {X 0,Y 208.003,Z 441.897,A -85,B 0,C 180,E1 -21302.863,E2 -21302.863} C_VEL
LIN {X 0,Y 204.026,Z 449.104,A -85,B 0,C 180,E1 -21306.665,E2 -21306.665} C_VEL
LIN {X 0,Y 200.798,Z 455.298,A -85,B 0,C 180,E1 -21310.915,E2 -21310.915} C_VEL
LIN {X 0,Y 199.47,Z 458.421,A -85,B 0,C 180,E1 -21313.63,E2 -21313.63} C_VEL
LIN {X 0,Y 198.105,Z 461.981,A -85,B 0,C 180,E1 -21317.712,E2 -21317.712} C_VEL
LIN {X 0,Y 197.561,Z 464.379,A -85,B 0,C 180,E1 -21321.821,E2 -21321.821} C_VEL
LIN {X 0,Y 197.506,Z 465.638,A -85,B 0,C 180,E1 -21325.92,E2 -21325.92} C_VEL
LIN {X 0,Y 197.619,Z 465.84,A -85,B 0,C 180,E1 -21327.963,E2 -21327.963} C_VEL
LIN {X 0,Y 197.654,Z 465.739,A -85,B 0,C 180,E1 -21330.001,E2 -21330.001} C_VEL
LIN {X 0,Y 197.632,Z 465.312,A -85,B 0,C 180,E1 -21332.039,E2 -21332.039} C_VEL
LIN {X 0,Y 197.602,Z 463.521,A -85,B 0,C 180,E1 -21336.126,E2 -21336.126} C_VEL
LIN {X 0,Y 197.807,Z 460.481,A -85,B 0,C 180,E1 -21340.234,E2 -21340.234} C_VEL
LIN {X 0,Y 198.742,Z 456.148,A -85,B 0,C 180,E1 -21344.333,E2 -21344.333} C_VEL
LIN {X 0,Y 200.421,Z 450.403,A -85,B 0,C 180,E1 -21348.398,E2 -21348.398} C_VEL
LIN {X 0,Y 202.989,Z 443.107,A -85,B 0,C 180,E1 -21352.388,E2 -21352.388} C_VEL
LIN {X 0,Y 206.06,Z 435.306,A -85,B 0,C 180,E1 -21355.778,E2 -21355.778} C_VEL
LIN {X 0,Y 209.643,Z 425.507,A -85,B 0,C 180,E1 -21359.222,E2 -21359.222} C_VEL
LIN {X 0,Y 213.885,Z 414.546,A -85,B 0,C 180,E1 -21362.275,E2 -21362.275} C_VEL
LIN {X 0,Y 218.044,Z 402.87,A -85,B 0,C 180,E1 -21364.899,E2 -21364.899} C_VEL
LIN {X 0,Y 221.18,Z 393.837,A -85,B 0,C 180,E1 -21366.57,E2 -21366.57} C_VEL
LIN {X 0,Y 221.295,Z 382.436,A -85,B 0,C 180,E1 -21368.847,E2 -21368.847} C_VEL
LIN {X 0,Y 220.599,Z 369.771,A -85,B 0,C 180,E1 -21371.178,E2 -21371.178} C_VEL
LIN {X 0,Y 218.822,Z 355.757,A -85,B 0,C 180,E1 -21373.589,E2 -21373.589} C_VEL
LIN {X 0,Y 216.054,Z 341.783,A -85,B 0,C 180,E1 -21375.863,E2 -21375.863} C_VEL
LIN {X 0,Y 213.289,Z 332.245,A -85,B 0,C 180,E1 -21377.426,E2 -21377.426} C_VEL
LIN {X 0,Y 209.398,Z 323.228,A -85,B 0,C 180,E1 -21379.118,E2 -21379.118} C_VEL
LIN {X 0,Y 206.397,Z 317.574,A -85,B 0,C 180,E1 -21380.291,E2 -21380.291} C_VEL
LIN {X 0,Y 204.18,Z 313.323,A -85,B 0,C 180,E1 -21381.134,E2 -21381.134} C_VEL
LIN {X 0,Y 202.336,Z 310.294,A -85,B 0,C 180,E1 -21381.822,E2 -21381.822} C_VEL
LIN {X 0,Y 201.793,Z 308.251,A -85,B 0,C 180,E1 -21382.148,E2 -21382.148} C_VEL
LIN {X 0,Y 201.173,Z 304.5,A -85,B 0,C 180,E1 -21386.978,E2 -21386.978} C_VEL
LIN {X 0,Y 200.722,Z 301.51,A -85,B 0,C 180,E1 -21391.087,E2 -21391.087} C_VEL
LIN {X 0,Y 200.226,Z 298.336,A -85,B 0,C 180,E1 -21395.871,E2 -21395.871} C_VEL
LIN {X 0,Y 199.795,Z 295.229,A -85,B 0,C 180,E1 -21401.009,E2 -21401.009} C_VEL
LIN {X 0,Y 199.843,Z 295.22,A -85,B 0,C 180,E1 -21405.747,E2 -21405.747} C_VEL
LIN {X 0,Y 200.029,Z 295.197,A -85,B 0,C 180,E1 -21409.88,E2 -21409.88} C_VEL
LIN {X 0,Y 200.02,Z 295.197,A -85,B 0,C 180,E1 -21413.947,E2 -21413.947} C_VEL
LIN {X 0,Y 200.325,Z 295.158,A -85,B 0,C 180,E1 -21417.987,E2 -21417.987} C_VEL
LIN {X 0,Y 200.485,Z 295.137,A -85,B 0,C 180,E1 -21419.998,E2 -21419.998} C_VEL
LIN {X 0,Y 200.034,Z 295.174,A -85,B 0,C 180,E1 -21424.027,E2 -21424.027} C_VEL
LIN {X 0,Y 200.136,Z 295.18,A -85,B 0,C 180,E1 -21428.072,E2 -21428.072} C_VEL
LIN {X 0,Y 200.072,Z 295.177,A -85,B 0,C 180,E1 -21430.395,E2 -21430.395} C_VEL
LIN {X 0,Y 199.808,Z 295.221,A -85,B 0,C 180,E1 -21436.341,E2 -21436.341} C_VEL
LIN {X 0,Y 199.702,Z 295.214,A -85,B 0,C 180,E1 -21440.603,E2 -21440.603} C_VEL
LIN {X 0,Y 199.674,Z 295.236,A -85,B 0,C 180,E1 -21444.981,E2 -21444.981} C_VEL
LIN {X 0,Y 199.665,Z 295.226,A -85,B 0,C 180,E1 -21449.521,E2 -21449.521} C_VEL
LIN {X 0,Y 199.658,Z 295.239,A -85,B 0,C 180,E1 -21452.347,E2 -21452.347} C_VEL
LIN {X 0,Y 199.639,Z 295.228,A -85,B 0,C 180,E1 -21456.756,E2 -21456.756} C_VEL
LIN {X 0,Y 199.639,Z 295.242,A -85,B 0,C 180,E1 -21459.318,E2 -21459.318} C_VEL
LIN {X 0,Y 199.629,Z 295.239,A -85,B 0,C 180,E1 -21464.754,E2 -21464.754} C_VEL
LIN {X 0,Y 199.662,Z 295.23,A -85,B 0,C 180,E1 -21468.025,E2 -21468.025} C_VEL
LIN {X 0,Y 199.676,Z 295.231,A -85,B 0,C 180,E1 -21470.74,E2 -21470.74} C_VEL
LIN {X 0,Y 199.63,Z 295.234,A -85,B 0,C 180,E1 -21475.715,E2 -21475.715} C_VEL
LIN {X 0,Y 199.699,Z 295.236,A -85,B 0,C 180,E1 -21478.135,E2 -21478.135} C_VEL
LIN {X 0,Y 199.682,Z 295.241,A -85,B 0,C 180,E1 -21482.77,E2 -21482.77} C_VEL
LIN {X 0,Y 199.732,Z 295.235,A -85,B 0,C 180,E1 -21487.227,E2 -21487.227} C_VEL
LIN {X 0,Y 199.764,Z 295.238,A -85,B 0,C 180,E1 -21491.06,E2 -21491.06} C_VEL
LIN {X 0,Y 200.734,Z 297.942,A -85,B 0,C 180,E1 -21491.524,E2 -21491.524} C_VEL
LIN {X 0,Y 202.807,Z 300.436,A -85,B 0,C 180,E1 -21492.295,E2 -21492.295} C_VEL
LIN {X 0,Y 204.617,Z 303.505,A -85,B 0,C 180,E1 -21493.04,E2 -21493.04} C_VEL
LIN {X 0,Y 210.686,Z 313.494,A -85,B 0,C 180,E1 -21495.535,E2 -21495.535} C_VEL
LIN {X 0,Y 216.234,Z 323.562,A -85,B 0,C 180,E1 -21497.968,E2 -21497.968} C_VEL
LIN {X 0,Y 220.431,Z 333.797,A -85,B 0,C 180,E1 -21500.205,E2 -21500.205} C_VEL
LIN {X 0,Y 222.114,Z 338.18,A -85,B 0,C 180,E1 -21501.185,E2 -21501.185} C_VEL
LIN {X 0,Y 224.849,Z 351.158,A -85,B 0,C 180,E1 -21503.8,E2 -21503.8} C_VEL
LIN {X 0,Y 226.093,Z 357.611,A -85,B 0,C 180,E1 -21505.202,E2 -21505.202} C_VEL
LIN {X 0,Y 222.842,Z 369.354,A -85,B 0,C 180,E1 -21507.061,E2 -21507.061} C_VEL
LIN {X 0,Y 219.098,Z 381.097,A -85,B 0,C 180,E1 -21509.31,E2 -21509.31} C_VEL
LIN {X 0,Y 215.272,Z 392.038,A -85,B 0,C 180,E1 -21511.87,E2 -21511.87} C_VEL
LIN {X 0,Y 211.55,Z 402.009,A -85,B 0,C 180,E1 -21514.729,E2 -21514.729} C_VEL
LIN {X 0,Y 207.699,Z 411.731,A -85,B 0,C 180,E1 -21518.163,E2 -21518.163} C_VEL
LIN {X 0,Y 204.493,Z 420.09,A -85,B 0,C 180,E1 -21521.899,E2 -21521.899} C_VEL
LIN {X 0,Y 202.215,Z 425.857,A -85,B 0,C 180,E1 -21525.107,E2 -21525.107} C_VEL
LIN {X 0,Y 200.305,Z 431.042,A -85,B 0,C 180,E1 -21528.686,E2 -21528.686} C_VEL
LIN {X 0,Y 198.701,Z 435.897,A -85,B 0,C 180,E1 -21533.138,E2 -21533.138} C_VEL
LIN {X 0,Y 197.694,Z 439.176,A -85,B 0,C 180,E1 -21537.524,E2 -21537.524} C_VEL
LIN {X 0,Y 197.345,Z 440.909,A -85,B 0,C 180,E1 -21541.278,E2 -21541.278} C_VEL
LIN {X 0,Y 197.407,Z 441.657,A -85,B 0,C 180,E1 -21545.036,E2 -21545.036} C_VEL
LIN {X 0,Y 198.069,Z 441.281,A -85,B 0,C 180,E1 -21549.692,E2 -21549.692} C_VEL
LIN {X 0,Y 198.762,Z 440.481,A -85,B 0,C 180,E1 -21552.206,E2 -21552.206} C_VEL
LIN {X 0,Y 199.909,Z 438.824,A -85,B 0,C 180,E1 -21555.326,E2 -21555.326} C_VEL
LIN {X 0,Y 202.335,Z 435.183,A -85,B 0,C 180,E1 -21559.83,E2 -21559.83} C_VEL
LIN {X 0,Y 205.009,Z 431.041,A -85,B 0,C 180,E1 -21563.459,E2 -21563.459} C_VEL
LIN {X 0,Y 208.769,Z 425.021,A -85,B 0,C 180,E1 -21567.413,E2 -21567.413} C_VEL
LIN {X 0,Y 213.169,Z 417.699,A -85,B 0,C 180,E1 -21571.083,E2 -21571.083} C_VEL
LIN {X 0,Y 218.105,Z 409.067,A -85,B 0,C 180,E1 -21574.451,E2 -21574.451} C_VEL
LIN {X 0,Y 222.719,Z 400.485,A -85,B 0,C 180,E1 -21577.151,E2 -21577.151} C_VEL
LIN {X 0,Y 228.088,Z 389.768,A -85,B 0,C 180,E1 -21579.84,E2 -21579.84} C_VEL
LIN {X 0,Y 233.513,Z 377.441,A -85,B 0,C 180,E1 -21582.322,E2 -21582.322} C_VEL
LIN {X 0,Y 236.581,Z 369.819,A -85,B 0,C 180,E1 -21583.577,E2 -21583.577} C_VEL
LIN {X 0,Y 236.716,Z 367.499,A -85,B 0,C 180,E1 -21584.159,E2 -21584.159} C_VEL
LIN {X 0,Y 235.882,Z 359.25,A -85,B 0,C 180,E1 -21586.542,E2 -21586.542} C_VEL
LIN {X 0,Y 234.606,Z 352.749,A -85,B 0,C 180,E1 -21588.555,E2 -21588.555} C_VEL
LIN {X 0,Y 232.855,Z 346.671,A -85,B 0,C 180,E1 -21590.633,E2 -21590.633} C_VEL
LIN {X 0,Y 229.632,Z 338.671,A -85,B 0,C 180,E1 -21593.853,E2 -21593.853} C_VEL
LIN {X 0,Y 226.977,Z 333.373,A -85,B 0,C 180,E1 -21596.452,E2 -21596.452} C_VEL
LIN {X 0,Y 225.154,Z 330.323,A -85,B 0,C 180,E1 -21598.213,E2 -21598.213} C_VEL
LIN {X 0,Y 223.643,Z 327.225,A -85,B 0,C 180,E1 -21600.002,E2 -21600.002} C_VEL
LIN {X 0,Y 221.028,Z 323.154,A -85,B 0,C 180,E1 -21603.125,E2 -21603.125} C_VEL
LIN {X 0,Y 218.054,Z 320.543,A -85,B 0,C 180,E1 -21607.222,E2 -21607.222} C_VEL
LIN {X 0,Y 217.287,Z 318.512,A -85,B 0,C 180,E1 -21609.309,E2 -21609.309} C_VEL
LIN {X 0,Y 215.493,Z 318.934,A -85,B 0,C 180,E1 -21615.853,E2 -21615.853} C_VEL
LIN {X 0,Y 216.11,Z 320.699,A -85,B 0,C 180,E1 -21620.591,E2 -21620.591} C_VEL
LIN {X 0,Y 217.35,Z 322.421,A -85,B 0,C 180,E1 -21623.589,E2 -21623.589} C_VEL
LIN {X 0,Y 218.738,Z 326.611,A -85,B 0,C 180,E1 -21626.605,E2 -21626.605} C_VEL
LIN {X 0,Y 220.751,Z 329.845,A -85,B 0,C 180,E1 -21629.309,E2 -21629.309} C_VEL
LIN {X 0,Y 222.267,Z 333.841,A -85,B 0,C 180,E1 -21631.383,E2 -21631.383} C_VEL
LIN {X 0,Y 223.697,Z 336.289,A -85,B 0,C 180,E1 -21632.839,E2 -21632.839} C_VEL
LIN {X 0,Y 224.861,Z 339.55,A -85,B 0,C 180,E1 -21634.237,E2 -21634.237} C_VEL
LIN {X 0,Y 225.832,Z 341.345,A -85,B 0,C 180,E1 -21635.153,E2 -21635.153} C_VEL
LIN {X 0,Y 229.753,Z 351.904,A -85,B 0,C 180,E1 -21639.144,E2 -21639.144} C_VEL
LIN {X 0,Y 231.116,Z 357.519,A -85,B 0,C 180,E1 -21640.829,E2 -21640.829} C_VEL
LIN {X 0,Y 231.912,Z 366.329,A -85,B 0,C 180,E1 -21642.992,E2 -21642.992} C_VEL
LIN {X 0,Y 232.07,Z 377.255,A -85,B 0,C 180,E1 -21645.5,E2 -21645.5} C_VEL
LIN {X 0,Y 231.32,Z 386.97,A -85,B 0,C 180,E1 -21647.681,E2 -21647.681} C_VEL
LIN {X 0,Y 229.659,Z 397.365,A -85,B 0,C 180,E1 -21650.013,E2 -21650.013} C_VEL
LIN {X 0,Y 228.757,Z 400.53,A -85,B 0,C 180,E1 -21650.704,E2 -21650.704} C_VEL
LIN {X 0,Y 223.05,Z 412.721,A -85,B 0,C 180,E1 -21653.227,E2 -21653.227} C_VEL
LIN {X 0,Y 217.484,Z 423.765,A -85,B 0,C 180,E1 -21656.123,E2 -21656.123} C_VEL
LIN {X 0,Y 215.881,Z 426.836,A -85,B 0,C 180,E1 -21657.062,E2 -21657.062} C_VEL
LIN {X 0,Y 213.447,Z 430.444,A -85,B 0,C 180,E1 -21658.146,E2 -21658.146} C_VEL
LIN {X 0,Y 208.007,Z 435.995,A -85,B 0,C 180,E1 -21659.815,E2 -21659.815} C_VEL
LIN {X 0,Y 202.646,Z 441.12,A -85,B 0,C 180,E1 -21661.647,E2 -21661.647} C_VEL
LIN {X 0,Y 200.386,Z 443.951,A -85,B 0,C 180,E1 -21662.971,E2 -21662.971} C_VEL
LIN {X 0,Y 196.587,Z 450.56,A -85,B 0,C 180,E1 -21666.845,E2 -21666.845} C_VEL
LIN {X 0,Y 193.614,Z 455.952,A -85,B 0,C 180,E1 -21670.933,E2 -21670.933} C_VEL
LIN {X 0,Y 191.758,Z 460.076,A -85,B 0,C 180,E1 -21675.136,E2 -21675.136} C_VEL
LIN {X 0,Y 190.702,Z 462.984,A -85,B 0,C 180,E1 -21679.383,E2 -21679.383} C_VEL
LIN {X 0,Y 190.411,Z 464.75,A -85,B 0,C 180,E1 -21683.644,E2 -21683.644} C_VEL
LIN {X 0,Y 190.437,Z 465.209,A -85,B 0,C 180,E1 -21685.769,E2 -21685.769} C_VEL
LIN {X 0,Y 190.528,Z 465.38,A -85,B 0,C 180,E1 -21687.888,E2 -21687.888} C_VEL
LIN {X 0,Y 190.589,Z 465.254,A -85,B 0,C 180,E1 -21690.001,E2 -21690.001} C_VEL
LIN {X 0,Y 190.545,Z 464.816,A -85,B 0,C 180,E1 -21692.115,E2 -21692.115} C_VEL
LIN {X 0,Y 190.513,Z 462.973,A -85,B 0,C 180,E1 -21696.355,E2 -21696.355} C_VEL
LIN {X 0,Y 190.768,Z 459.869,A -85,B 0,C 180,E1 -21700.616,E2 -21700.616} C_VEL
LIN {X 0,Y 191.81,Z 455.469,A -85,B 0,C 180,E1 -21704.863,E2 -21704.863} C_VEL
LIN {X 0,Y 193.607,Z 449.647,A -85,B 0,C 180,E1 -21709.07,E2 -21709.07} C_VEL
LIN {X 0,Y 196.345,Z 442.268,A -85,B 0,C 180,E1 -21713.189,E2 -21713.189} C_VEL
LIN {X 0,Y 199.585,Z 434.374,A -85,B 0,C 180,E1 -21716.679,E2 -21716.679} C_VEL
LIN {X 0,Y 203.03,Z 425.33,A -85,B 0,C 180,E1 -21719.941,E2 -21719.941} C_VEL
LIN {X 0,Y 207.145,Z 415.178,A -85,B 0,C 180,E1 -21722.879,E2 -21722.879} C_VEL
LIN {X 0,Y 211.413,Z 403.701,A -85,B 0,C 180,E1 -21725.575,E2 -21725.575} C_VEL
LIN {X 0,Y 214.555,Z 395.023,A -85,B 0,C 180,E1 -21727.243,E2 -21727.243} C_VEL
LIN {X 0,Y 214.925,Z 385.238,A -85,B 0,C 180,E1 -21729.315,E2 -21729.315} C_VEL
LIN {X 0,Y 214.472,Z 372.14,A -85,B 0,C 180,E1 -21731.873,E2 -21731.873} C_VEL
LIN {X 0,Y 213.006,Z 359.035,A -85,B 0,C 180,E1 -21734.254,E2 -21734.254} C_VEL
LIN {X 0,Y 210.662,Z 345.894,A -85,B 0,C 180,E1 -21736.521,E2 -21736.521} C_VEL
LIN {X 0,Y 208.109,Z 336.009,A -85,B 0,C 180,E1 -21738.245,E2 -21738.245} C_VEL
LIN {X 0,Y 204.282,Z 327.025,A -85,B 0,C 180,E1 -21740.069,E2 -21740.069} C_VEL
LIN {X 0,Y 199.701,Z 317.951,A -85,B 0,C 180,E1 -21742.039,E2 -21742.039} C_VEL
LIN {X 0,Y 197.651,Z 314.108,A -85,B 0,C 180,E1 -21742.883,E2 -21742.883} C_VEL
LIN {X 0,Y 196.521,Z 312.31,A -85,B 0,C 180,E1 -21743.339,E2 -21743.339} C_VEL
LIN {X 0,Y 194.858,Z 309.239,A -85,B 0,C 180,E1 -21744.038,E2 -21744.038} C_VEL
LIN {X 0,Y 194.444,Z 307.676,A -85,B 0,C 180,E1 -21744.348,E2 -21744.348} C_VEL
LIN {X 0,Y 194.152,Z 305.591,A -85,B 0,C 180,E1 -21747.111,E2 -21747.111} C_VEL
LIN {X 0,Y 193.653,Z 302.306,A -85,B 0,C 180,E1 -21751.847,E2 -21751.847} C_VEL
LIN {X 0,Y 193.204,Z 299.396,A -85,B 0,C 180,E1 -21756.411,E2 -21756.411} C_VEL
LIN {X 0,Y 192.818,Z 296.491,A -85,B 0,C 180,E1 -21761.386,E2 -21761.386} C_VEL
LIN {X 0,Y 192.761,Z 296.1,A -85,B 0,C 180,E1 -21762.212,E2 -21762.212} C_VEL
LIN {X 0,Y 192.812,Z 296.097,A -85,B 0,C 180,E1 -21767.365,E2 -21767.365} C_VEL
LIN {X 0,Y 193.037,Z 296.068,A -85,B 0,C 180,E1 -21771.624,E2 -21771.624} C_VEL
LIN {X 0,Y 193.266,Z 296.037,A -85,B 0,C 180,E1 -21777.914,E2 -21777.914} C_VEL
LIN {X 0,Y 193.449,Z 296.013,A -85,B 0,C 180,E1 -21779.998,E2 -21779.998} C_VEL
LIN {X 0,Y 192.981,Z 296.052,A -85,B 0,C 180,E1 -21784.175,E2 -21784.175} C_VEL
LIN {X 0,Y 193.083,Z 296.059,A -85,B 0,C 180,E1 -21788.369,E2 -21788.369} C_VEL
LIN {X 0,Y 193.014,Z 296.055,A -85,B 0,C 180,E1 -21790.536,E2 -21790.536} C_VEL
LIN {X 0,Y 192.761,Z 296.096,A -85,B 0,C 180,E1 -21796.956,E2 -21796.956} C_VEL
LIN {X 0,Y 192.638,Z 296.098,A -85,B 0,C 180,E1 -21801.394,E2 -21801.394} C_VEL
LIN {X 0,Y 192.666,Z 296.112,A -85,B 0,C 180,E1 -21804.222,E2 -21804.222} C_VEL
LIN {X 0,Y 192.644,Z 296.095,A -85,B 0,C 180,E1 -21808.886,E2 -21808.886} C_VEL
LIN {X 0,Y 192.598,Z 296.118,A -85,B 0,C 180,E1 -21813.183,E2 -21813.183} C_VEL
LIN {X 0,Y 192.573,Z 296.119,A -85,B 0,C 180,E1 -21818.343,E2 -21818.343} C_VEL
LIN {X 0,Y 192.537,Z 296.108,A -85,B 0,C 180,E1 -21823.108,E2 -21823.108} C_VEL
LIN {X 0,Y 192.597,Z 296.118,A -85,B 0,C 180,E1 -21826.867,E2 -21826.867} C_VEL
LIN {X 0,Y 192.596,Z 296.118,A -85,B 0,C 180,E1 -21831.657,E2 -21831.657} C_VEL
LIN {X 0,Y 192.596,Z 296.119,A -85,B 0,C 180,E1 -21836.812,E2 -21836.812} C_VEL
LIN {X 0,Y 192.659,Z 296.111,A -85,B 0,C 180,E1 -21841.69,E2 -21841.69} C_VEL
LIN {X 0,Y 192.7,Z 296.109,A -85,B 0,C 180,E1 -21846.346,E2 -21846.346} C_VEL
LIN {X 0,Y 192.682,Z 296.235,A -85,B 0,C 180,E1 -21848.969,E2 -21848.969} C_VEL
LIN {X 0,Y 193.552,Z 298.755,A -85,B 0,C 180,E1 -21849.428,E2 -21849.428} C_VEL
LIN {X 0,Y 195.83,Z 301.469,A -85,B 0,C 180,E1 -21850.367,E2 -21850.367} C_VEL
LIN {X 0,Y 197.69,Z 304.577,A -85,B 0,C 180,E1 -21851.2,E2 -21851.2} C_VEL
LIN {X 0,Y 199.03,Z 306.55,A -85,B 0,C 180,E1 -21851.761,E2 -21851.761} C_VEL
LIN {X 0,Y 203.941,Z 314.713,A -85,B 0,C 180,E1 -21853.945,E2 -21853.945} C_VEL
LIN {X 0,Y 210.214,Z 326.084,A -85,B 0,C 180,E1 -21856.905,E2 -21856.905} C_VEL
LIN {X 0,Y 213.331,Z 333.229,A -85,B 0,C 180,E1 -21858.598,E2 -21858.598} C_VEL
LIN {X 0,Y 216.518,Z 342.213,A -85,B 0,C 180,E1 -21860.659,E2 -21860.659} C_VEL
LIN {X 0,Y 219.213,Z 355.974,A -85,B 0,C 180,E1 -21863.625,E2 -21863.625} C_VEL
LIN {X 0,Y 219.793,Z 359.801,A -85,B 0,C 180,E1 -21864.494,E2 -21864.494} C_VEL
LIN {X 0,Y 216.068,Z 371.964,A -85,B 0,C 180,E1 -21866.502,E2 -21866.502} C_VEL
LIN {X 0,Y 211.945,Z 384.187,A -85,B 0,C 180,E1 -21869.003,E2 -21869.003} C_VEL
LIN {X 0,Y 207.656,Z 395.758,A -85,B 0,C 180,E1 -21871.938,E2 -21871.938} C_VEL
LIN {X 0,Y 203.671,Z 405.847,A -85,B 0,C 180,E1 -21875.119,E2 -21875.119} C_VEL
LIN {X 0,Y 199.946,Z 414.855,A -85,B 0,C 180,E1 -21878.649,E2 -21878.649} C_VEL
LIN {X 0,Y 196.881,Z 422.415,A -85,B 0,C 180,E1 -21882.366,E2 -21882.366} C_VEL
LIN {X 0,Y 194.669,Z 427.916,A -85,B 0,C 180,E1 -21885.708,E2 -21885.708} C_VEL
LIN {X 0,Y 193.023,Z 432.419,A -85,B 0,C 180,E1 -21889.127,E2 -21889.127} C_VEL
LIN {X 0,Y 191.489,Z 436.752,A -85,B 0,C 180,E1 -21893.437,E2 -21893.437} C_VEL
LIN {X 0,Y 190.579,Z 439.748,A -85,B 0,C 180,E1 -21897.748,E2 -21897.748} C_VEL
LIN {X 0,Y 190.24,Z 441.466,A -85,B 0,C 180,E1 -21901.828,E2 -21901.828} C_VEL
LIN {X 0,Y 190.416,Z 442.151,A -85,B 0,C 180,E1 -21906.193,E2 -21906.193} C_VEL
LIN {X 0,Y 190.914,Z 441.875,A -85,B 0,C 180,E1 -21909.375,E2 -21909.375} C_VEL
LIN {X 0,Y 192.263,Z 440.367,A -85,B 0,C 180,E1 -21913.987,E2 -21913.987} C_VEL
LIN {X 0,Y 193.382,Z 438.885,A -85,B 0,C 180,E1 -21916.621,E2 -21916.621} C_VEL
LIN {X 0,Y 195.704,Z 435.675,A -85,B 0,C 180,E1 -21920.625,E2 -21920.625} C_VEL
LIN {X 0,Y 198.659,Z 431.426,A -85,B 0,C 180,E1 -21924.454,E2 -21924.454} C_VEL
LIN {X 0,Y 202.897,Z 425.043,A -85,B 0,C 180,E1 -21928.699,E2 -21928.699} C_VEL
LIN {X 0,Y 207.749,Z 417.385,A -85,B 0,C 180,E1 -21932.56,E2 -21932.56} C_VEL
LIN {X 0,Y 212.328,Z 409.885,A -85,B 0,C 180,E1 -21935.535,E2 -21935.535} C_VEL
LIN {X 0,Y 217.873,Z 400.012,A -85,B 0,C 180,E1 -21938.654,E2 -21938.654} C_VEL
LIN {X 0,Y 223.395,Z 389.379,A -85,B 0,C 180,E1 -21941.309,E2 -21941.309} C_VEL
LIN {X 0,Y 228.366,Z 378.675,A -85,B 0,C 180,E1 -21943.488,E2 -21943.488} C_VEL
LIN {X 0,Y 231.102,Z 372.336,A -85,B 0,C 180,E1 -21944.57,E2 -21944.57} C_VEL
LIN {X 0,Y 231.24,Z 368.963,A -85,B 0,C 180,E1 -21945.481,E2 -21945.481} C_VEL
LIN {X 0,Y 230.409,Z 360.529,A -85,B 0,C 180,E1 -21948.12,E2 -21948.12} C_VEL
LIN {X 0,Y 228.825,Z 352.988,A -85,B 0,C 180,E1 -21950.723,E2 -21950.723} C_VEL
LIN {X 0,Y 226.188,Z 345.431,A -85,B 0,C 180,E1 -21953.859,E2 -21953.859} C_VEL
LIN {X 0,Y 224,Z 340.218,A -85,B 0,C 180,E1 -21956.404,E2 -21956.404} C_VEL
LIN {X 0,Y 220.952,Z 334.258,A -85,B 0,C 180,E1 -21960.002,E2 -21960.002} C_VEL
LIN {X 0,Y 218.316,Z 329.438,A -85,B 0,C 180,E1 -21963.693,E2 -21963.693} C_VEL
LIN {X 0,Y 215.893,Z 327.357,A -85,B 0,C 180,E1 -21967.295,E2 -21967.295} C_VEL
LIN {X 0,Y 215.247,Z 325.42,A -85,B 0,C 180,E1 -21969.398,E2 -21969.398} C_VEL
LIN {X 0,Y 213.622,Z 325.661,A -85,B 0,C 180,E1 -21975.262,E2 -21975.262} C_VEL
LIN {X 0,Y 214.064,Z 327.374,A -85,B 0,C 180,E1 -21980.167,E2 -21980.167} C_VEL
LIN {X 0,Y 215.158,Z 329.053,A -85,B 0,C 180,E1 -21983.19,E2 -21983.19} C_VEL
LIN {X 0,Y 216.318,Z 333.155,A -85,B 0,C 180,E1 -21986.255,E2 -21986.255} C_VEL
LIN {X 0,Y 218.051,Z 336.41,A -85,B 0,C 180,E1 -21988.914,E2 -21988.914} C_VEL
LIN {X 0,Y 219.284,Z 339.943,A -85,B 0,C 180,E1 -21990.852,E2 -21990.852} C_VEL
LIN {X 0,Y 220.451,Z 342.204,A -85,B 0,C 180,E1 -21992.243,E2 -21992.243} C_VEL
LIN {X 0,Y 222.701,Z 348.491,A -85,B 0,C 180,E1 -21995.111,E2 -21995.111} C_VEL
LIN {X 0,Y 225.181,Z 355.888,A -85,B 0,C 180,E1 -21998.056,E2 -21998.056} C_VEL
LIN {X 0,Y 226.295,Z 360.275,A -85,B 0,C 180,E1 -21999.544,E2 -21999.544} C_VEL
LIN {X 0,Y 226.963,Z 368.516,A -85,B 0,C 180,E1 -22001.743,E2 -22001.743} C_VEL
LIN {X 0,Y 226.724,Z 379.902,A -85,B 0,C 180,E1 -22004.526,E2 -22004.526} C_VEL
LIN {X 0,Y 225.748,Z 389.451,A -85,B 0,C 180,E1 -22006.774,E2 -22006.774} C_VEL
LIN {X 0,Y 223.585,Z 400.182,A -85,B 0,C 180,E1 -22009.336,E2 -22009.336} C_VEL
LIN {X 0,Y 220.123,Z 407.852,A -85,B 0,C 180,E1 -22010.91,E2 -22010.91} C_VEL
LIN {X 0,Y 214.028,Z 419.615,A -85,B 0,C 180,E1 -22013.769,E2 -22013.769} C_VEL
LIN {X 0,Y 208.597,Z 429.466,A -85,B 0,C 180,E1 -22016.807,E2 -22016.807} C_VEL
LIN {X 0,Y 203.928,Z 437.736,A -85,B 0,C 180,E1 -22020.021,E2 -22020.021} C_VEL
LIN {X 0,Y 200.386,Z 443.951,A -85,B 0,C 180,E1 -22022.971,E2 -22022.971} C_VEL
LIN {X 0,Y 198.166,Z 446.672,A -85,B 0,C 180,E1 -22024.351,E2 -22024.351} C_VEL
LIN {X 0,Y 193.053,Z 450.688,A -85,B 0,C 180,E1 -22026.55,E2 -22026.55} C_VEL
LIN {X 0,Y 188.279,Z 454.227,A -85,B 0,C 180,E1 -22028.932,E2 -22028.932} C_VEL
LIN {X 0,Y 186.639,Z 456.1,A -85,B 0,C 180,E1 -22030.565,E2 -22030.565} C_VEL
LIN {X 0,Y 184.827,Z 459.812,A -85,B 0,C 180,E1 -22034.565,E2 -22034.565} C_VEL
LIN {X 0,Y 183.667,Z 462.65,A -85,B 0,C 180,E1 -22038.971,E2 -22038.971} C_VEL
LIN {X 0,Y 183.322,Z 464.351,A -85,B 0,C 180,E1 -22043.397,E2 -22043.397} C_VEL
LIN {X 0,Y 183.361,Z 464.78,A -85,B 0,C 180,E1 -22045.605,E2 -22045.605} C_VEL
LIN {X 0,Y 183.526,Z 464.764,A -85,B 0,C 180,E1 -22050.002,E2 -22050.002} C_VEL
LIN {X 0,Y 183.43,Z 463.523,A -85,B 0,C 180,E1 -22054.396,E2 -22054.396} C_VEL
LIN {X 0,Y 183.476,Z 460.987,A -85,B 0,C 180,E1 -22058.815,E2 -22058.815} C_VEL
LIN {X 0,Y 184.183,Z 457.175,A -85,B 0,C 180,E1 -22063.237,E2 -22063.237} C_VEL
LIN {X 0,Y 185.724,Z 452.006,A -85,B 0,C 180,E1 -22067.623,E2 -22067.623} C_VEL
LIN {X 0,Y 188.178,Z 445.35,A -85,B 0,C 180,E1 -22071.932,E2 -22071.932} C_VEL
LIN {X 0,Y 191.092,Z 438.16,A -85,B 0,C 180,E1 -22075.605,E2 -22075.605} C_VEL
LIN {X 0,Y 194.757,Z 429.515,A -85,B 0,C 180,E1 -22079.156,E2 -22079.156} C_VEL
LIN {X 0,Y 198.373,Z 420.738,A -85,B 0,C 180,E1 -22082.103,E2 -22082.103} C_VEL
LIN {X 0,Y 202.613,Z 410.412,A -85,B 0,C 180,E1 -22084.915,E2 -22084.915} C_VEL
LIN {X 0,Y 207.208,Z 398.065,A -85,B 0,C 180,E1 -22087.628,E2 -22087.628} C_VEL
LIN {X 0,Y 208.295,Z 394.529,A -85,B 0,C 180,E1 -22088.311,E2 -22088.311} C_VEL
LIN {X 0,Y 208.513,Z 382.915,A -85,B 0,C 180,E1 -22090.867,E2 -22090.867} C_VEL
LIN {X 0,Y 208.008,Z 370.663,A -85,B 0,C 180,E1 -22093.331,E2 -22093.331} C_VEL
LIN {X 0,Y 206.406,Z 356.469,A -85,B 0,C 180,E1 -22096.006,E2 -22096.006} C_VEL
LIN {X 0,Y 204.125,Z 344.395,A -85,B 0,C 180,E1 -22098.203,E2 -22098.203} C_VEL
LIN {X 0,Y 201.716,Z 336.563,A -85,B 0,C 180,E1 -22099.726,E2 -22099.726} C_VEL
LIN {X 0,Y 197.194,Z 326.607,A -85,B 0,C 180,E1 -22101.98,E2 -22101.98} C_VEL
LIN {X 0,Y 194.611,Z 321.561,A -85,B 0,C 180,E1 -22103.181,E2 -22103.181} C_VEL
LIN {X 0,Y 192.482,Z 317.451,A -85,B 0,C 180,E1 -22104.171,E2 -22104.171} C_VEL
LIN {X 0,Y 190.404,Z 313.492,A -85,B 0,C 180,E1 -22105.1,E2 -22105.1} C_VEL
LIN {X 0,Y 187.801,Z 309.309,A -85,B 0,C 180,E1 -22106.253,E2 -22106.253} C_VEL
LIN {X 0,Y 187.182,Z 307.097,A -85,B 0,C 180,E1 -22106.691,E2 -22106.691} C_VEL
LIN {X 0,Y 186.772,Z 304.368,A -85,B 0,C 180,E1 -22110.711,E2 -22110.711} C_VEL
LIN {X 0,Y 186.331,Z 301.319,A -85,B 0,C 180,E1 -22115.485,E2 -22115.485} C_VEL
LIN {X 0,Y 185.906,Z 298.194,A -85,B 0,C 180,E1 -22120.93,E2 -22120.93} C_VEL
LIN {X 0,Y 185.715,Z 296.979,A -85,B 0,C 180,E1 -22123.509,E2 -22123.509} C_VEL
LIN {X 0,Y 185.895,Z 296.958,A -85,B 0,C 180,E1 -22129.416,E2 -22129.416} C_VEL
LIN {X 0,Y 185.947,Z 296.95,A -85,B 0,C 180,E1 -22133.487,E2 -22133.487} C_VEL
LIN {X 0,Y 186.21,Z 296.916,A -85,B 0,C 180,E1 -22137.835,E2 -22137.835} C_VEL
LIN {X 0,Y 186.412,Z 296.89,A -85,B 0,C 180,E1 -22139.998,E2 -22139.998} C_VEL
LIN {X 0,Y 185.928,Z 296.929,A -85,B 0,C 180,E1 -22144.333,E2 -22144.333} C_VEL
LIN {X 0,Y 186.033,Z 296.935,A -85,B 0,C 180,E1 -22148.689,E2 -22148.689} C_VEL
LIN {X 0,Y 185.738,Z 296.954,A -85,B 0,C 180,E1 -22153.12,E2 -22153.12} C_VEL
LIN {X 0,Y 185.693,Z 296.974,A -85,B 0,C 180,E1 -22157.622,E2 -22157.622} C_VEL
LIN {X 0,Y 185.598,Z 296.981,A -85,B 0,C 180,E1 -22162.248,E2 -22162.248} C_VEL
LIN {X 0,Y 185.561,Z 296.979,A -85,B 0,C 180,E1 -22167.029,E2 -22167.029} C_VEL
LIN {X 0,Y 185.578,Z 296.978,A -85,B 0,C 180,E1 -22169.49,E2 -22169.49} C_VEL
LIN {X 0,Y 185.509,Z 296.987,A -85,B 0,C 180,E1 -22174.627,E2 -22174.627} C_VEL
LIN {X 0,Y 185.543,Z 296.986,A -85,B 0,C 180,E1 -22177.301,E2 -22177.301} C_VEL
LIN {X 0,Y 185.493,Z 297,A -85,B 0,C 180,E1 -22180.73,E2 -22180.73} C_VEL
LIN {X 0,Y 185.551,Z 296.998,A -85,B 0,C 180,E1 -22186.021,E2 -22186.021} C_VEL
LIN {X 0,Y 185.537,Z 296.984,A -85,B 0,C 180,E1 -22189.911,E2 -22189.911} C_VEL
LIN {X 0,Y 185.556,Z 296.996,A -85,B 0,C 180,E1 -22192.697,E2 -22192.697} C_VEL
LIN {X 0,Y 185.54,Z 297.001,A -85,B 0,C 180,E1 -22197.973,E2 -22197.973} C_VEL
LIN {X 0,Y 185.577,Z 296.986,A -85,B 0,C 180,E1 -22200.573,E2 -22200.573} C_VEL
LIN {X 0,Y 185.581,Z 296.988,A -85,B 0,C 180,E1 -22205.38,E2 -22205.38} C_VEL
LIN {X 0,Y 185.643,Z 297.06,A -85,B 0,C 180,E1 -22206.687,E2 -22206.687} C_VEL
LIN {X 0,Y 186.541,Z 299.721,A -85,B 0,C 180,E1 -22207.212,E2 -22207.212} C_VEL
LIN {X 0,Y 188.789,Z 302.359,A -85,B 0,C 180,E1 -22208.219,E2 -22208.219} C_VEL
LIN {X 0,Y 190.559,Z 305.412,A -85,B 0,C 180,E1 -22209.084,E2 -22209.084} C_VEL
LIN {X 0,Y 192.1,Z 307.436,A -85,B 0,C 180,E1 -22209.759,E2 -22209.759} C_VEL
LIN {X 0,Y 197.115,Z 315.596,A -85,B 0,C 180,E1 -22212.181,E2 -22212.181} C_VEL
LIN {X 0,Y 203.381,Z 327.074,A -85,B 0,C 180,E1 -22215.356,E2 -22215.356} C_VEL
LIN {X 0,Y 207.1,Z 334.973,A -85,B 0,C 180,E1 -22217.429,E2 -22217.429} C_VEL
LIN {X 0,Y 210.608,Z 345.053,A -85,B 0,C 180,E1 -22219.884,E2 -22219.884} C_VEL
LIN {X 0,Y 212.942,Z 357.919,A -85,B 0,C 180,E1 -22222.811,E2 -22222.811} C_VEL
LIN {X 0,Y 213.522,Z 361.17,A -85,B 0,C 180,E1 -22223.598,E2 -22223.598} C_VEL
LIN {X 0,Y 209.314,Z 374.514,A -85,B 0,C 180,E1 -22225.916,E2 -22225.916} C_VEL
LIN {X 0,Y 205.235,Z 386.035,A -85,B 0,C 180,E1 -22228.406,E2 -22228.406} C_VEL
LIN {X 0,Y 201.405,Z 395.897,A -85,B 0,C 180,E1 -22230.998,E2 -22230.998} C_VEL
LIN {X 0,Y 197.302,Z 405.845,A -85,B 0,C 180,E1 -22234.191,E2 -22234.191} C_VEL
LIN {X 0,Y 193.385,Z 414.954,A -85,B 0,C 180,E1 -22237.831,E2 -22237.831} C_VEL
LIN {X 0,Y 190.139,Z 422.684,A -85,B 0,C 180,E1 -22241.728,E2 -22241.728} C_VEL
LIN {X 0,Y 187.785,Z 428.23,A -85,B 0,C 180,E1 -22245.186,E2 -22245.186} C_VEL
LIN {X 0,Y 185.914,Z 433.18,A -85,B 0,C 180,E1 -22249.09,E2 -22249.09} C_VEL
LIN {X 0,Y 184.277,Z 437.595,A -85,B 0,C 180,E1 -22253.756,E2 -22253.756} C_VEL
LIN {X 0,Y 183.412,Z 440.437,A -85,B 0,C 180,E1 -22258.204,E2 -22258.204} C_VEL
LIN {X 0,Y 183.144,Z 442.043,A -85,B 0,C 180,E1 -22262.494,E2 -22262.494} C_VEL
LIN {X 0,Y 183.367,Z 442.609,A -85,B 0,C 180,E1 -22266.406,E2 -22266.406} C_VEL
LIN {X 0,Y 184.057,Z 442.23,A -85,B 0,C 180,E1 -22270.474,E2 -22270.474} C_VEL
LIN {X 0,Y 185.092,Z 441.204,A -85,B 0,C 180,E1 -22273.831,E2 -22273.831} C_VEL
LIN {X 0,Y 187.309,Z 438.524,A -85,B 0,C 180,E1 -22278.624,E2 -22278.624} C_VEL
LIN {X 0,Y 189.979,Z 435.079,A -85,B 0,C 180,E1 -22282.635,E2 -22282.635} C_VEL
LIN {X 0,Y 193.823,Z 429.813,A -85,B 0,C 180,E1 -22287.054,E2 -22287.054} C_VEL
LIN {X 0,Y 198.089,Z 423.743,A -85,B 0,C 180,E1 -22290.848,E2 -22290.848} C_VEL
LIN {X 0,Y 202.78,Z 416.669,A -85,B 0,C 180,E1 -22294.301,E2 -22294.301} C_VEL
LIN {X 0,Y 208.641,Z 407.385,A -85,B 0,C 180,E1 -22297.835,E2 -22297.835} C_VEL
LIN {X 0,Y 214.133,Z 397.914,A -85,B 0,C 180,E1 -22300.678,E2 -22300.678} C_VEL
LIN {X 0,Y 220.07,Z 386.703,A -85,B 0,C 180,E1 -22303.342,E2 -22303.342} C_VEL
LIN {X 0,Y 225.496,Z 375.046,A -85,B 0,C 180,E1 -22305.564,E2 -22305.564} C_VEL
LIN {X 0,Y 225.906,Z 372.913,A -85,B 0,C 180,E1 -22306.12,E2 -22306.12} C_VEL
LIN {X 0,Y 225.413,Z 364.874,A -85,B 0,C 180,E1 -22308.765,E2 -22308.765} C_VEL
LIN {X 0,Y 224.108,Z 357.232,A -85,B 0,C 180,E1 -22311.577,E2 -22311.577} C_VEL
LIN {X 0,Y 222.029,Z 350.541,A -85,B 0,C 180,E1 -22314.553,E2 -22314.553} C_VEL
LIN {X 0,Y 220.014,Z 345.345,A -85,B 0,C 180,E1 -22317.256,E2 -22317.256} C_VEL
LIN {X 0,Y 217.134,Z 339.227,A -85,B 0,C 180,E1 -22321.305,E2 -22321.305} C_VEL
LIN {X 0,Y 215.713,Z 336.223,A -85,B 0,C 180,E1 -22323.738,E2 -22323.738} C_VEL
LIN {X 0,Y 213.396,Z 333.909,A -85,B 0,C 180,E1 -22327.572,E2 -22327.572} C_VEL
LIN {X 0,Y 212.931,Z 332.257,A -85,B 0,C 180,E1 -22329.501,E2 -22329.501} C_VEL
LIN {X 0,Y 211.689,Z 332.223,A -85,B 0,C 180,E1 -22333.44,E2 -22333.44} C_VEL
LIN {X 0,Y 211.455,Z 333.024,A -85,B 0,C 180,E1 -22337.407,E2 -22337.407} C_VEL
LIN {X 0,Y 212.508,Z 335.136,A -85,B 0,C 180,E1 -22342.183,E2 -22342.183} C_VEL
LIN {X 0,Y 214.882,Z 342.023,A -85,B 0,C 180,E1 -22347.988,E2 -22347.988} C_VEL
LIN {X 0,Y 217.119,Z 348.242,A -85,B 0,C 180,E1 -22351.738,E2 -22351.738} C_VEL
LIN {X 0,Y 219.057,Z 354.461,A -85,B 0,C 180,E1 -22354.683,E2 -22354.683} C_VEL
LIN {X 0,Y 221.145,Z 361.645,A -85,B 0,C 180,E1 -22357.661,E2 -22357.661} C_VEL
LIN {X 0,Y 221.924,Z 366.587,A -85,B 0,C 180,E1 -22359.301,E2 -22359.301} C_VEL
LIN {X 0,Y 221.929,Z 375.454,A -85,B 0,C 180,E1 -22361.686,E2 -22361.686} C_VEL
LIN {X 0,Y 221.081,Z 385.952,A -85,B 0,C 180,E1 -22364.378,E2 -22364.378} C_VEL
LIN {X 0,Y 219.172,Z 396.727,A -85,B 0,C 180,E1 -22367.048,E2 -22367.048} C_VEL
LIN {X 0,Y 217.589,Z 402.607,A -85,B 0,C 180,E1 -22368.511,E2 -22368.511} C_VEL
LIN {X 0,Y 211.861,Z 413.578,A -85,B 0,C 180,E1 -22370.931,E2 -22370.931} C_VEL
LIN {X 0,Y 205.832,Z 424.296,A -85,B 0,C 180,E1 -22373.917,E2 -22373.917} C_VEL
LIN {X 0,Y 200.325,Z 433.568,A -85,B 0,C 180,E1 -22377.18,E2 -22377.18} C_VEL
LIN {X 0,Y 195.37,Z 441.92,A -85,B 0,C 180,E1 -22380.948,E2 -22380.948} C_VEL
LIN {X 0,Y 190.96,Z 448.915,A -85,B 0,C 180,E1 -22384.962,E2 -22384.962} C_VEL
LIN {X 0,Y 187.472,Z 454.659,A -85,B 0,C 180,E1 -22389.253,E2 -22389.253} C_VEL
LIN {X 0,Y 186.639,Z 456.1,A -85,B 0,C 180,E1 -22390.565,E2 -22390.565} C_VEL
LIN {X 0,Y 185.141,Z 457.84,A -85,B 0,C 180,E1 -22392.248,E2 -22392.248} C_VEL
LIN {X 0,Y 181.13,Z 460.178,A -85,B 0,C 180,E1 -22394.989,E2 -22394.989} C_VEL
LIN {X 0,Y 178.013,Z 461.661,A -85,B 0,C 180,E1 -22397.282,E2 -22397.282} C_VEL
LIN {X 0,Y 176.606,Z 462.601,A -85,B 0,C 180,E1 -22399.12,E2 -22399.12} C_VEL
LIN {X 0,Y 176.437,Z 462.835,A -85,B 0,C 180,E1 -22399.753,E2 -22399.753} C_VEL
LIN {X 0,Y 176.235,Z 463.955,A -85,B 0,C 180,E1 -22403.131,E2 -22403.131} C_VEL
LIN {X 0,Y 176.306,Z 464.353,A -85,B 0,C 180,E1 -22405.429,E2 -22405.429} C_VEL
LIN {X 0,Y 176.463,Z 464.274,A -85,B 0,C 180,E1 -22410.002,E2 -22410.002} C_VEL
LIN {X 0,Y 176.355,Z 462.973,A -85,B 0,C 180,E1 -22414.573,E2 -22414.573} C_VEL
LIN {X 0,Y 176.418,Z 460.397,A -85,B 0,C 180,E1 -22419.171,E2 -22419.171} C_VEL
LIN {X 0,Y 177.216,Z 456.516,A -85,B 0,C 180,E1 -22423.767,E2 -22423.767} C_VEL
LIN {X 0,Y 178.897,Z 451.272,A -85,B 0,C 180,E1 -22428.319,E2 -22428.319} C_VEL
LIN {X 0,Y 181.516,Z 444.534,A -85,B 0,C 180,E1 -22432.781,E2 -22432.781} C_VEL
LIN {X 0,Y 184.632,Z 437.256,A -85,B 0,C 180,E1 -22436.57,E2 -22436.57} C_VEL
LIN {X 0,Y 188.485,Z 428.505,A -85,B 0,C 180,E1 -22440.225,E2 -22440.225} C_VEL
LIN {X 0,Y 192.311,Z 419.609,A -85,B 0,C 180,E1 -22443.243,E2 -22443.243} C_VEL
LIN {X 0,Y 196.743,Z 409.154,A -85,B 0,C 180,E1 -22446.117,E2 -22446.117} C_VEL
LIN {X 0,Y 201.126,Z 397.795,A -85,B 0,C 180,E1 -22448.655,E2 -22448.655} C_VEL
LIN {X 0,Y 201.85,Z 395.338,A -85,B 0,C 180,E1 -22449.15,E2 -22449.15} C_VEL
LIN {X 0,Y 202.166,Z 384.097,A -85,B 0,C 180,E1 -22451.749,E2 -22451.749} C_VEL
LIN {X 0,Y 201.872,Z 372.828,A -85,B 0,C 180,E1 -22454.131,E2 -22454.131} C_VEL
LIN {X 0,Y 200.556,Z 359,A -85,B 0,C 180,E1 -22456.895,E2 -22456.895} C_VEL
LIN {X 0,Y 198.306,Z 346.164,A -85,B 0,C 180,E1 -22459.365,E2 -22459.365} C_VEL
LIN {X 0,Y 195.87,Z 338.826,A -85,B 0,C 180,E1 -22460.967,E2 -22460.967} C_VEL
LIN {X 0,Y 191.149,Z 328.058,A -85,B 0,C 180,E1 -22463.555,E2 -22463.555} C_VEL
LIN {X 0,Y 187.721,Z 321.567,A -85,B 0,C 180,E1 -22465.264,E2 -22465.264} C_VEL
LIN {X 0,Y 185.505,Z 317.252,A -85,B 0,C 180,E1 -22466.406,E2 -22466.406} C_VEL
LIN {X 0,Y 183.437,Z 313.363,A -85,B 0,C 180,E1 -22467.436,E2 -22467.436} C_VEL
LIN {X 0,Y 182.726,Z 312.045,A -85,B 0,C 180,E1 -22467.793,E2 -22467.793} C_VEL
LIN {X 0,Y 180.616,Z 308.896,A -85,B 0,C 180,E1 -22468.802,E2 -22468.802} C_VEL
LIN {X 0,Y 179.891,Z 306.577,A -85,B 0,C 180,E1 -22469.263,E2 -22469.263} C_VEL
LIN {X 0,Y 179.422,Z 303.277,A -85,B 0,C 180,E1 -22474.475,E2 -22474.475} C_VEL
LIN {X 0,Y 179.019,Z 300.499,A -85,B 0,C 180,E1 -22479.307,E2 -22479.307} C_VEL
LIN {X 0,Y 178.668,Z 297.933,A -85,B 0,C 180,E1 -22484.308,E2 -22484.308} C_VEL
LIN {X 0,Y 178.84,Z 297.837,A -85,B 0,C 180,E1 -22489.255,E2 -22489.255} C_VEL
LIN {X 0,Y 178.911,Z 297.827,A -85,B 0,C 180,E1 -22493.23,E2 -22493.23} C_VEL
LIN {X 0,Y 179.155,Z 297.795,A -85,B 0,C 180,E1 -22497.749,E2 -22497.749} C_VEL
LIN {X 0,Y 179.375,Z 297.766,A -85,B 0,C 180,E1 -22499.998,E2 -22499.998} C_VEL
LIN {X 0,Y 178.877,Z 297.806,A -85,B 0,C 180,E1 -22504.504,E2 -22504.504} C_VEL
LIN {X 0,Y 178.982,Z 297.813,A -85,B 0,C 180,E1 -22509.034,E2 -22509.034} C_VEL
LIN {X 0,Y 178.665,Z 297.838,A -85,B 0,C 180,E1 -22513.649,E2 -22513.649} C_VEL
LIN {X 0,Y 178.625,Z 297.839,A -85,B 0,C 180,E1 -22519.213,E2 -22519.213} C_VEL
LIN {X 0,Y 178.536,Z 297.869,A -85,B 0,C 180,E1 -22525.121,E2 -22525.121} C_VEL
LIN {X 0,Y 178.477,Z 297.874,A -85,B 0,C 180,E1 -22530.788,E2 -22530.788} C_VEL
LIN {X 0,Y 178.49,Z 297.864,A -85,B 0,C 180,E1 -22534.219,E2 -22534.219} C_VEL
LIN {X 0,Y 178.421,Z 297.884,A -85,B 0,C 180,E1 -22539.064,E2 -22539.064} C_VEL
LIN {X 0,Y 178.422,Z 297.867,A -85,B 0,C 180,E1 -22542.034,E2 -22542.034} C_VEL
LIN {X 0,Y 178.46,Z 297.877,A -85,B 0,C 180,E1 -22545.139,E2 -22545.139} C_VEL
LIN {X 0,Y 178.498,Z 297.862,A -85,B 0,C 180,E1 -22548.421,E2 -22548.421} C_VEL
LIN {X 0,Y 178.455,Z 297.873,A -85,B 0,C 180,E1 -22553.789,E2 -22553.789} C_VEL
LIN {X 0,Y 178.487,Z 297.872,A -85,B 0,C 180,E1 -22556.545,E2 -22556.545} C_VEL
LIN {X 0,Y 178.518,Z 297.865,A -85,B 0,C 180,E1 -22560.004,E2 -22560.004} C_VEL
LIN {X 0,Y 178.497,Z 297.926,A -85,B 0,C 180,E1 -22564.099,E2 -22564.099} C_VEL
LIN {X 0,Y 179.473,Z 300.641,A -85,B 0,C 180,E1 -22564.708,E2 -22564.708} C_VEL
LIN {X 0,Y 181.855,Z 303.195,A -85,B 0,C 180,E1 -22565.867,E2 -22565.867} C_VEL
LIN {X 0,Y 183.628,Z 306.388,A -85,B 0,C 180,E1 -22566.846,E2 -22566.846} C_VEL
LIN {X 0,Y 185.027,Z 308.166,A -85,B 0,C 180,E1 -22567.52,E2 -22567.52} C_VEL
LIN {X 0,Y 187.203,Z 311.517,A -85,B 0,C 180,E1 -22568.656,E2 -22568.656} C_VEL
LIN {X 0,Y 192.327,Z 320.004,A -85,B 0,C 180,E1 -22571.334,E2 -22571.334} C_VEL
LIN {X 0,Y 198.456,Z 331.714,A -85,B 0,C 180,E1 -22574.759,E2 -22574.759} C_VEL
LIN {X 0,Y 201.624,Z 338.675,A -85,B 0,C 180,E1 -22576.706,E2 -22576.706} C_VEL
LIN {X 0,Y 204.785,Z 348.203,A -85,B 0,C 180,E1 -22579.163,E2 -22579.163} C_VEL
LIN {X 0,Y 206.884,Z 360.821,A -85,B 0,C 180,E1 -22582.189,E2 -22582.189} C_VEL
LIN {X 0,Y 207.117,Z 363.554,A -85,B 0,C 180,E1 -22582.838,E2 -22582.838} C_VEL
LIN {X 0,Y 202.598,Z 376.88,A -85,B 0,C 180,E1 -22585.273,E2 -22585.273} C_VEL
LIN {X 0,Y 198.199,Z 388.645,A -85,B 0,C 180,E1 -22587.967,E2 -22587.967} C_VEL
LIN {X 0,Y 193.767,Z 399.477,A -85,B 0,C 180,E1 -22591.038,E2 -22591.038} C_VEL
LIN {X 0,Y 189.783,Z 408.661,A -85,B 0,C 180,E1 -22594.246,E2 -22594.246} C_VEL
LIN {X 0,Y 185.727,Z 417.618,A -85,B 0,C 180,E1 -22598.156,E2 -22598.156} C_VEL
LIN {X 0,Y 182.535,Z 424.961,A -85,B 0,C 180,E1 -22602.224,E2 -22602.224} C_VEL
LIN {X 0,Y 180.258,Z 430.142,A -85,B 0,C 180,E1 -22605.836,E2 -22605.836} C_VEL
LIN {X 0,Y 178.68,Z 434.154,A -85,B 0,C 180,E1 -22609.277,E2 -22609.277} C_VEL
LIN {X 0,Y 177.096,Z 438.401,A -85,B 0,C 180,E1 -22614.12,E2 -22614.12} C_VEL
LIN {X 0,Y 176.257,Z 441.119,A -85,B 0,C 180,E1 -22618.698,E2 -22618.698} C_VEL
LIN {X 0,Y 176.057,Z 442.575,A -85,B 0,C 180,E1 -22623.045,E2 -22623.045} C_VEL
LIN {X 0,Y 176.351,Z 443.057,A -85,B 0,C 180,E1 -22627.156,E2 -22627.156} C_VEL
LIN {X 0,Y 177.467,Z 442.381,A -85,B 0,C 180,E1 -22632.315,E2 -22632.315} C_VEL
LIN {X 0,Y 178.476,Z 441.392,A -85,B 0,C 180,E1 -22635.135,E2 -22635.135} C_VEL
LIN {X 0,Y 180.022,Z 439.679,A -85,B 0,C 180,E1 -22638.423,E2 -22638.423} C_VEL
LIN {X 0,Y 183.466,Z 435.631,A -85,B 0,C 180,E1 -22643.554,E2 -22643.554} C_VEL
LIN {X 0,Y 186.8,Z 431.324,A -85,B 0,C 180,E1 -22647.389,E2 -22647.389} C_VEL
LIN {X 0,Y 191.648,Z 424.948,A -85,B 0,C 180,E1 -22651.653,E2 -22651.653} C_VEL
LIN {X 0,Y 196.992,Z 417.449,A -85,B 0,C 180,E1 -22655.477,E2 -22655.477} C_VEL
LIN {X 0,Y 203.15,Z 408.246,A -85,B 0,C 180,E1 -22659.074,E2 -22659.074} C_VEL
LIN {X 0,Y 208.837,Z 398.929,A -85,B 0,C 180,E1 -22661.932,E2 -22661.932} C_VEL
LIN {X 0,Y 214.697,Z 388.48,A -85,B 0,C 180,E1 -22664.483,E2 -22664.483} C_VEL
LIN {X 0,Y 220.508,Z 376.732,A -85,B 0,C 180,E1 -22666.798,E2 -22666.798} C_VEL
LIN {X 0,Y 220.383,Z 369.155,A -85,B 0,C 180,E1 -22669.436,E2 -22669.436} C_VEL
LIN {X 0,Y 219.53,Z 362.107,A -85,B 0,C 180,E1 -22672.182,E2 -22672.182} C_VEL
LIN {X 0,Y 217.755,Z 355.356,A -85,B 0,C 180,E1 -22675.374,E2 -22675.374} C_VEL
LIN {X 0,Y 216.035,Z 350.431,A -85,B 0,C 180,E1 -22678.138,E2 -22678.138} C_VEL
LIN {X 0,Y 213.78,Z 345.146,A -85,B 0,C 180,E1 -22681.886,E2 -22681.886} C_VEL
LIN {X 0,Y 212.825,Z 342.883,A -85,B 0,C 180,E1 -22683.789,E2 -22683.789} C_VEL
LIN {X 0,Y 210.752,Z 340.501,A -85,B 0,C 180,E1 -22687.667,E2 -22687.667} C_VEL
LIN {X 0,Y 210.376,Z 338.933,A -85,B 0,C 180,E1 -22689.617,E2 -22689.617} C_VEL
LIN {X 0,Y 209.232,Z 338.907,A -85,B 0,C 180,E1 -22693.601,E2 -22693.601} C_VEL
LIN {X 0,Y 209.035,Z 339.788,A -85,B 0,C 180,E1 -22697.615,E2 -22697.615} C_VEL
LIN {X 0,Y 209.82,Z 341.54,A -85,B 0,C 180,E1 -22701.622,E2 -22701.622} C_VEL
LIN {X 0,Y 211.842,Z 348.411,A -85,B 0,C 180,E1 -22707.677,E2 -22707.677} C_VEL
LIN {X 0,Y 213.582,Z 354.059,A -85,B 0,C 180,E1 -22711.183,E2 -22711.183} C_VEL
LIN {X 0,Y 215.536,Z 361.46,A -85,B 0,C 180,E1 -22714.797,E2 -22714.797} C_VEL
LIN {X 0,Y 216.911,Z 367.509,A -85,B 0,C 180,E1 -22717.333,E2 -22717.333} C_VEL
LIN {X 0,Y 217.218,Z 371.015,A -85,B 0,C 180,E1 -22718.525,E2 -22718.525} C_VEL
LIN {X 0,Y 216.796,Z 379.67,A -85,B 0,C 180,E1 -22720.97,E2 -22720.97} C_VEL
LIN {X 0,Y 215.454,Z 390.184,A -85,B 0,C 180,E1 -22723.785,E2 -22723.785} C_VEL
LIN {X 0,Y 213.075,Z 400.608,A -85,B 0,C 180,E1 -22726.524,E2 -22726.524} C_VEL
LIN {X 0,Y 211.634,Z 404.627,A -85,B 0,C 180,E1 -22727.543,E2 -22727.543} C_VEL
LIN {X 0,Y 205.456,Z 415.632,A -85,B 0,C 180,E1 -22730.107,E2 -22730.107} C_VEL
LIN {X 0,Y 199.288,Z 425.912,A -85,B 0,C 180,E1 -22733.167,E2 -22733.167} C_VEL
LIN {X 0,Y 193.018,Z 435.702,A -85,B 0,C 180,E1 -22736.897,E2 -22736.897} C_VEL
LIN {X 0,Y 187.884,Z 443.77,A -85,B 0,C 180,E1 -22740.905,E2 -22740.905} C_VEL
LIN {X 0,Y 183.487,Z 450.32,A -85,B 0,C 180,E1 -22745.083,E2 -22745.083} C_VEL
LIN {X 0,Y 180.003,Z 455.656,A -85,B 0,C 180,E1 -22749.567,E2 -22749.567} C_VEL
LIN {X 0,Y 177.923,Z 459.525,A -85,B 0,C 180,E1 -22753.95,E2 -22753.95} C_VEL
LIN {X 0,Y 176.627,Z 462.327,A -85,B 0,C 180,E1 -22758.526,E2 -22758.526} C_VEL
LIN {X 0,Y 176.437,Z 462.835,A -85,B 0,C 180,E1 -22759.753,E2 -22759.753} C_VEL
LIN {X 0,Y 175.59,Z 463.541,A -85,B 0,C 180,E1 -22761.644,E2 -22761.644} C_VEL
LIN {X 0,Y 172.625,Z 464.065,A -85,B 0,C 180,E1 -22764.755,E2 -22764.755} C_VEL
LIN {X 0,Y 170.283,Z 464.072,A -85,B 0,C 180,E1 -22767.318,E2 -22767.318} C_VEL
LIN {X 0,Y 169.408,Z 463.896,A -85,B 0,C 180,E1 -22769.312,E2 -22769.312} C_VEL
LIN {X 0,Y 169.399,Z 463.779,A -85,B 0,C 180,E1 -22769.986,E2 -22769.986} C_VEL
LIN {X 0,Y 169.33,Z 462.283,A -85,B 0,C 180,E1 -22775.031,E2 -22775.031} C_VEL
LIN {X 0,Y 169.358,Z 459.772,A -85,B 0,C 180,E1 -22779.556,E2 -22779.556} C_VEL
LIN {X 0,Y 170.258,Z 455.828,A -85,B 0,C 180,E1 -22784.341,E2 -22784.341} C_VEL
LIN {X 0,Y 172.1,Z 450.5,A -85,B 0,C 180,E1 -22789.07,E2 -22789.07} C_VEL
LIN {X 0,Y 174.895,Z 443.668,A -85,B 0,C 180,E1 -22793.695,E2 -22793.695} C_VEL
LIN {X 0,Y 178.8,Z 435.166,A -85,B 0,C 180,E1 -22798.145,E2 -22798.145} C_VEL
LIN {X 0,Y 182.83,Z 426.041,A -85,B 0,C 180,E1 -22801.909,E2 -22801.909} C_VEL
LIN {X 0,Y 187.817,Z 415.116,A -85,B 0,C 180,E1 -22805.452,E2 -22805.452} C_VEL
LIN {X 0,Y 192.531,Z 403.86,A -85,B 0,C 180,E1 -22808.358,E2 -22808.358} C_VEL
LIN {X 0,Y 195.414,Z 396.23,A -85,B 0,C 180,E1 -22810.008,E2 -22810.008} C_VEL
LIN {X 0,Y 195.917,Z 383.971,A -85,B 0,C 180,E1 -22812.968,E2 -22812.968} C_VEL
LIN {X 0,Y 195.723,Z 373.943,A -85,B 0,C 180,E1 -22815.194,E2 -22815.194} C_VEL
LIN {X 0,Y 194.544,Z 360.29,A -85,B 0,C 180,E1 -22818.06,E2 -22818.06} C_VEL
LIN {X 0,Y 192.782,Z 349.122,A -85,B 0,C 180,E1 -22820.356,E2 -22820.356} C_VEL
LIN {X 0,Y 190.344,Z 341.594,A -85,B 0,C 180,E1 -22822.13,E2 -22822.13} C_VEL
LIN {X 0,Y 186.084,Z 331.857,A -85,B 0,C 180,E1 -22824.665,E2 -22824.665} C_VEL
LIN {X 0,Y 181.277,Z 322.09,A -85,B 0,C 180,E1 -22827.379,E2 -22827.379} C_VEL
LIN {X 0,Y 178.697,Z 317.09,A -85,B 0,C 180,E1 -22828.813,E2 -22828.813} C_VEL
LIN {X 0,Y 176.469,Z 313.286,A -85,B 0,C 180,E1 -22830,E2 -22830} C_VEL
LIN {X 0,Y 175.742,Z 311.781,A -85,B 0,C 180,E1 -22830.418,E2 -22830.418} C_VEL
LIN {X 0,Y 173.556,Z 308.732,A -85,B 0,C 180,E1 -22831.586,E2 -22831.586} C_VEL
LIN {X 0,Y 172.607,Z 305.916,A -85,B 0,C 180,E1 -22832.242,E2 -22832.242} C_VEL
LIN {X 0,Y 172.289,Z 303.739,A -85,B 0,C 180,E1 -22835.923,E2 -22835.923} C_VEL
LIN {X 0,Y 171.967,Z 301.066,A -85,B 0,C 180,E1 -22840.914,E2 -22840.914} C_VEL
LIN {X 0,Y 171.603,Z 298.738,A -85,B 0,C 180,E1 -22845.773,E2 -22845.773} C_VEL
LIN {X 0,Y 171.852,Z 298.708,A -85,B 0,C 180,E1 -22850.583,E2 -22850.583} C_VEL
LIN {X 0,Y 171.815,Z 298.71,A -85,B 0,C 180,E1 -22855.305,E2 -22855.305} C_VEL
LIN {X 0,Y 172.338,Z 298.643,A -85,B 0,C 180,E1 -22859.998,E2 -22859.998} C_VEL
LIN {X 0,Y 171.827,Z 298.684,A -85,B 0,C 180,E1 -22864.69,E2 -22864.69} C_VEL
LIN {X 0,Y 171.907,Z 298.692,A -85,B 0,C 180,E1 -22869.409,E2 -22869.409} C_VEL
LIN {X 0,Y 171.582,Z 298.725,A -85,B 0,C 180,E1 -22874.224,E2 -22874.224} C_VEL
LIN {X 0,Y 171.546,Z 298.718,A -85,B 0,C 180,E1 -22879.559,E2 -22879.559} C_VEL
LIN {X 0,Y 171.47,Z 298.745,A -85,B 0,C 180,E1 -22885.613,E2 -22885.613} C_VEL
LIN {X 0,Y 171.439,Z 298.747,A -85,B 0,C 180,E1 -22890.582,E2 -22890.582} C_VEL
LIN {X 0,Y 171.4,Z 298.74,A -85,B 0,C 180,E1 -22895.029,E2 -22895.029} C_VEL
LIN {X 0,Y 171.382,Z 298.761,A -85,B 0,C 180,E1 -22898.815,E2 -22898.815} C_VEL
LIN {X 0,Y 171.366,Z 298.749,A -85,B 0,C 180,E1 -22904.198,E2 -22904.198} C_VEL
LIN {X 0,Y 171.415,Z 298.741,A -85,B 0,C 180,E1 -22909.003,E2 -22909.003} C_VEL
LIN {X 0,Y 171.433,Z 298.757,A -85,B 0,C 180,E1 -22912.051,E2 -22912.051} C_VEL
LIN {X 0,Y 171.415,Z 298.762,A -85,B 0,C 180,E1 -22917.79,E2 -22917.79} C_VEL
LIN {X 0,Y 171.437,Z 298.757,A -85,B 0,C 180,E1 -22921.212,E2 -22921.212} C_VEL
LIN {X 0,Y 172.292,Z 301.304,A -85,B 0,C 180,E1 -22921.836,E2 -22921.836} C_VEL
LIN {X 0,Y 174.135,Z 303.457,A -85,B 0,C 180,E1 -22922.873,E2 -22922.873} C_VEL
LIN {X 0,Y 174.909,Z 304.31,A -85,B 0,C 180,E1 -22923.293,E2 -22923.293} C_VEL
LIN {X 0,Y 176.8,Z 307.459,A -85,B 0,C 180,E1 -22924.406,E2 -22924.406} C_VEL
LIN {X 0,Y 178.251,Z 309.247,A -85,B 0,C 180,E1 -22925.172,E2 -22925.172} C_VEL
LIN {X 0,Y 180.473,Z 312.718,A -85,B 0,C 180,E1 -22926.451,E2 -22926.451} C_VEL
LIN {X 0,Y 185.844,Z 321.438,A -85,B 0,C 180,E1 -22929.499,E2 -22929.499} C_VEL
LIN {X 0,Y 191.507,Z 332.256,A -85,B 0,C 180,E1 -22932.926,E2 -22932.926} C_VEL
LIN {X 0,Y 195.801,Z 341.498,A -85,B 0,C 180,E1 -22935.714,E2 -22935.714} C_VEL
LIN {X 0,Y 198.954,Z 351.337,A -85,B 0,C 180,E1 -22938.41,E2 -22938.41} C_VEL
LIN {X 0,Y 200.824,Z 363.769,A -85,B 0,C 180,E1 -22941.565,E2 -22941.565} C_VEL
LIN {X 0,Y 200.853,Z 365.325,A -85,B 0,C 180,E1 -22941.953,E2 -22941.953} C_VEL
LIN {X 0,Y 196.322,Z 378.015,A -85,B 0,C 180,E1 -22944.349,E2 -22944.349} C_VEL
LIN {X 0,Y 192.168,Z 388.716,A -85,B 0,C 180,E1 -22946.854,E2 -22946.854} C_VEL
LIN {X 0,Y 187.543,Z 399.606,A -85,B 0,C 180,E1 -22949.999,E2 -22949.999} C_VEL
LIN {X 0,Y 183.073,Z 409.494,A -85,B 0,C 180,E1 -22953.569,E2 -22953.569} C_VEL
LIN {X 0,Y 179.196,Z 417.719,A -85,B 0,C 180,E1 -22957.266,E2 -22957.266} C_VEL
LIN {X 0,Y 175.778,Z 425.213,A -85,B 0,C 180,E1 -22961.53,E2 -22961.53} C_VEL
LIN {X 0,Y 173.367,Z 430.423,A -85,B 0,C 180,E1 -22965.275,E2 -22965.275} C_VEL
LIN {X 0,Y 171.448,Z 435.068,A -85,B 0,C 180,E1 -22969.479,E2 -22969.479} C_VEL
LIN {X 0,Y 169.902,Z 439.154,A -85,B 0,C 180,E1 -22974.498,E2 -22974.498} C_VEL
LIN {X 0,Y 169.047,Z 442.005,A -85,B 0,C 180,E1 -22979.925,E2 -22979.925} C_VEL
LIN {X 0,Y 168.975,Z 443.127,A -85,B 0,C 180,E1 -22983.718,E2 -22983.718} C_VEL
LIN {X 0,Y 169.453,Z 443.495,A -85,B 0,C 180,E1 -22988.469,E2 -22988.469} C_VEL
LIN {X 0,Y 170.275,Z 443.093,A -85,B 0,C 180,E1 -22992.022,E2 -22992.022} C_VEL
LIN {X 0,Y 172.278,Z 441.298,A -85,B 0,C 180,E1 -22997.245,E2 -22997.245} C_VEL
LIN {X 0,Y 174.824,Z 438.611,A -85,B 0,C 180,E1 -23001.617,E2 -23001.617} C_VEL
LIN {X 0,Y 178.773,Z 434.095,A -85,B 0,C 180,E1 -23006.611,E2 -23006.611} C_VEL
LIN {X 0,Y 183.967,Z 427.846,A -85,B 0,C 180,E1 -23011.477,E2 -23011.477} C_VEL
LIN {X 0,Y 188.785,Z 421.619,A -85,B 0,C 180,E1 -23015.091,E2 -23015.091} C_VEL
LIN {X 0,Y 194.157,Z 414.324,A -85,B 0,C 180,E1 -23018.412,E2 -23018.412} C_VEL
LIN {X 0,Y 200.135,Z 405.569,A -85,B 0,C 180,E1 -23021.578,E2 -23021.578} C_VEL
LIN {X 0,Y 206.428,Z 395.521,A -85,B 0,C 180,E1 -23024.435,E2 -23024.435} C_VEL
LIN {X 0,Y 212.697,Z 384.273,A -85,B 0,C 180,E1 -23026.968,E2 -23026.968} C_VEL
LIN {X 0,Y 214.969,Z 379.853,A -85,B 0,C 180,E1 -23027.829,E2 -23027.829} C_VEL
LIN {X 0,Y 215.31,Z 377.136,A -85,B 0,C 180,E1 -23028.708,E2 -23028.708} C_VEL
LIN {X 0,Y 215.215,Z 370.99,A -85,B 0,C 180,E1 -23031.079,E2 -23031.079} C_VEL
LIN {X 0,Y 214.575,Z 365.582,A -85,B 0,C 180,E1 -23033.419,E2 -23033.419} C_VEL
LIN {X 0,Y 213.325,Z 360.08,A -85,B 0,C 180,E1 -23036.224,E2 -23036.224} C_VEL
LIN {X 0,Y 211.938,Z 355.469,A -85,B 0,C 180,E1 -23039.052,E2 -23039.052} C_VEL
LIN {X 0,Y 209.95,Z 350.054,A -85,B 0,C 180,E1 -23043.251,E2 -23043.251} C_VEL
LIN {X 0,Y 209.694,Z 349.385,A -85,B 0,C 180,E1 -23043.845,E2 -23043.845} C_VEL
LIN {X 0,Y 207.865,Z 346.972,A -85,B 0,C 180,E1 -23047.775,E2 -23047.775} C_VEL
LIN {X 0,Y 207.582,Z 345.47,A -85,B 0,C 180,E1 -23049.748,E2 -23049.748} C_VEL
LIN {X 0,Y 206.497,Z 345.491,A -85,B 0,C 180,E1 -23053.785,E2 -23053.785} C_VEL
LIN {X 0,Y 206.339,Z 346.456,A -85,B 0,C 180,E1 -23057.853,E2 -23057.853} C_VEL
LIN {X 0,Y 206.644,Z 347.282,A -85,B 0,C 180,E1 -23059.885,E2 -23059.885} C_VEL
